C07284=1038.998,375.277,369.594,173.156,44.214,158.680
C07285=1039.007,375.523,369.554,173.163,44.217,158.682
C07286=1039.015,375.770,369.513,173.170,44.221,158.684
C07287=1039.023,376.016,369.472,173.177,44.225,158.685
C07288=1039.032,376.263,369.431,173.184,44.229,158.687
C07289=1039.040,376.510,369.390,173.191,44.233,158.688
C07290=1039.049,376.756,369.350,173.199,44.237,158.690
C07291=1039.062,377.144,369.286,173.210,44.244,158.693
C07292=1039.076,377.532,369.222,173.221,44.250,158.695
C07293=1039.089,377.920,369.157,173.233,44.256,158.698
C07294=1039.103,378.308,369.092,173.244,44.263,158.701
C07295=1039.111,378.555,369.051,173.251,44.266,158.702
C07296=1039.119,378.802,369.011,173.259,44.270,158.704
C07297=1039.128,379.048,368.969,173.266,44.275,158.706
C07298=1039.136,379.295,368.928,173.273,44.279,158.707
C07299=1039.145,379.541,368.886,173.280,44.283,158.709
C07300=1039.153,379.787,368.845,173.288,44.287,158.711
C07301=1039.161,380.034,368.804,173.295,44.291,158.712
C07302=1039.170,380.280,368.762,173.302,44.296,158.714
C07303=1039.178,380.526,368.721,173.309,44.300,158.716
C07304=1039.187,380.773,368.679,173.317,44.304,158.718
C07305=1039.195,381.018,368.638,173.324,44.308,158.719
C07306=1039.204,381.265,368.597,173.331,44.312,158.721
C07307=1039.213,381.512,368.555,173.339,44.317,158.723
C07308=1039.221,381.758,368.514,173.346,44.321,158.725
C07309=1039.230,382.004,368.472,173.354,44.325,158.726
C07310=1039.238,382.251,368.430,173.361,44.329,158.728
C07311=1039.247,382.498,368.389,173.369,44.334,158.730
C07312=1039.255,382.743,368.347,173.376,44.338,158.732
C07313=1039.264,382.990,368.305,173.383,44.343,158.733
C07314=1039.273,383.236,368.264,173.391,44.347,158.735
C07315=1039.281,383.483,368.221,173.399,44.351,158.737
C07316=1039.289,383.728,368.180,173.406,44.355,158.739
C07317=1039.298,383.975,368.138,173.414,44.360,158.741
C07318=1039.307,384.221,368.097,173.421,44.364,158.742
C07319=1039.316,384.467,368.055,173.429,44.369,158.744
C07320=1039.325,384.713,368.012,173.437,44.373,158.746
C07321=1039.334,384.960,367.970,173.445,44.378,158.748
C07322=1039.343,385.206,367.928,173.452,44.382,158.750
C07323=1039.351,385.453,367.887,173.460,44.387,158.752
C07324=1039.360,385.699,367.845,173.468,44.391,158.754
C07325=1039.368,385.944,367.802,173.475,44.395,158.755
C07326=1039.377,386.191,367.761,173.483,44.400,158.757
C07327=1039.386,386.437,367.719,173.491,44.405,158.759
C07328=1039.395,386.683,367.677,173.498,44.409,158.761
C07329=1039.404,386.929,367.634,173.506,44.414,158.763
C07330=1039.413,387.176,367.592,173.515,44.418,158.765
C07331=1039.422,387.422,367.550,173.522,44.423,158.767
C07332=1039.431,387.669,367.508,173.531,44.427,158.769
C07333=1039.440,387.915,367.465,173.538,44.432,158.770
C07334=1039.449,388.161,367.423,173.546,44.437,158.772
C07335=1039.458,388.407,367.381,173.554,44.441,158.774
C07336=1039.466,388.653,367.338,173.562,44.446,158.776
C07337=1039.476,388.899,367.295,173.570,44.450,158.778
C07338=1039.484,389.145,367.253,173.578,44.455,158.780
C07339=1039.493,389.391,367.211,173.585,44.460,158.782
C07340=1039.502,389.638,367.167,173.594,44.464,158.784
C07341=1039.512,389.883,367.125,173.601,44.469,158.786
C07342=1039.520,390.129,367.082,173.610,44.474,158.788
C07343=1039.529,390.376,367.040,173.618,44.479,158.790
C07344=1039.537,390.622,366.997,173.626,44.483,158.792
C07345=1039.547,390.868,366.954,173.634,44.489,158.794
C07346=1039.556,391.114,366.911,173.643,44.493,158.796
C07347=1039.565,391.352,366.870,173.650,44.498,158.798
C07348=1039.573,391.589,366.828,173.658,44.502,158.800
C07349=1039.582,391.827,366.786,173.666,44.507,158.802
C07350=1039.591,392.065,366.745,173.674,44.512,158.804
C07351=1039.599,392.303,366.703,173.682,44.517,158.806
C07352=1039.608,392.541,366.662,173.690,44.521,158.808
C07353=1039.617,392.779,366.620,173.698,44.526,158.809
C07354=1039.626,393.017,366.578,173.707,44.531,158.812
C07355=1039.634,393.263,366.535,173.714,44.536,158.813
C07356=1039.643,393.510,366.492,173.723,44.541,158.816
C07357=1039.653,393.755,366.449,173.732,44.546,158.818
C07358=1039.662,394.001,366.405,173.740,44.551,158.820
C07359=1039.671,394.247,366.362,173.748,44.555,158.822
C07360=1039.681,394.493,366.319,173.756,44.561,158.824
C07361=1039.689,394.739,366.275,173.765,44.566,158.826
C07362=1039.699,394.986,366.232,173.774,44.571,158.828
C07363=1039.708,395.231,366.188,173.783,44.576,158.830
C07364=1039.717,395.477,366.145,173.790,44.581,158.832
C07365=1039.726,395.723,366.101,173.799,44.586,158.834
C07366=1039.735,395.969,366.057,173.808,44.591,158.837
C07367=1039.744,396.214,366.013,173.816,44.596,158.839
C07368=1039.754,396.461,365.971,173.825,44.602,158.841
C07369=1039.763,396.706,365.927,173.834,44.607,158.843
C07370=1039.772,396.952,365.883,173.843,44.612,158.845
C07371=1039.781,397.198,365.839,173.851,44.617,158.847
C07372=1039.790,397.444,365.795,173.860,44.623,158.850
C07373=1039.800,397.690,365.751,173.868,44.628,158.852
C07374=1039.809,397.936,365.707,173.877,44.632,158.854
C07375=1039.819,398.181,365.664,173.886,44.638,158.856
C07376=1039.828,398.427,365.619,173.894,44.643,158.858
C07377=1039.837,398.673,365.576,173.903,44.649,158.861
C07378=1039.846,398.919,365.532,173.912,44.654,158.863
C07379=1039.856,399.165,365.488,173.921,44.659,158.865
C07380=1039.865,399.411,365.443,173.930,44.664,158.867
C07381=1039.875,399.657,365.399,173.939,44.670,158.870
C07382=1039.884,399.903,365.354,173.948,44.675,158.872
C07383=1039.893,400.148,365.311,173.957,44.680,158.874
C07384=1039.903,400.395,365.267,173.966,44.686,158.876
C07385=1039.912,400.640,365.222,173.975,44.691,158.879
C07386=1039.922,400.886,365.178,173.985,44.697,158.881
C07387=1039.931,401.132,365.133,173.994,44.702,158.883
C07388=1039.941,401.378,365.089,174.003,44.708,158.886
C07389=1039.951,401.623,365.044,174.012,44.714,158.888
C07390=1039.960,401.869,365.000,174.021,44.719,158.890
C07391=1039.970,402.115,364.955,174.030,44.725,158.893
C07392=1039.979,402.361,364.910,174.039,44.730,158.895
C07393=1039.989,402.607,364.866,174.049,44.736,158.897
C07394=1039.999,402.852,364.821,174.058,44.741,158.900
C07395=1040.008,403.098,364.776,174.067,44.747,158.902
C07396=1040.017,403.344,364.732,174.076,44.753,158.905
C07397=1040.027,403.590,364.687,174.085,44.758,158.907
C07398=1040.036,403.835,364.642,174.094,44.764,158.909
C07399=1040.045,404.054,364.602,174.103,44.769,158.911
C07400=1040.053,404.274,364.561,174.111,44.774,158.914
C07401=1040.062,404.493,364.521,174.119,44.779,158.916
C07402=1040.071,404.711,364.481,174.128,44.784,158.918
C07403=1040.079,404.930,364.441,174.136,44.789,158.920
C07404=1040.088,405.150,364.400,174.145,44.794,158.922
C07405=1040.096,405.369,364.360,174.153,44.800,158.924
C07406=1040.105,405.588,364.319,174.162,44.805,158.927
C07407=1040.114,405.809,364.279,174.171,44.810,158.929
C07408=1040.122,406.030,364.238,174.179,44.816,158.931
C07409=1040.131,406.251,364.198,174.188,44.820,158.933
C07410=1040.140,406.473,364.157,174.196,44.826,158.936
C07411=1040.149,406.693,364.117,174.205,44.831,158.938
C07412=1040.158,406.914,364.075,174.214,44.837,158.940
C07413=1040.166,407.136,364.034,174.222,44.842,158.942
C07414=1040.175,407.356,363.994,174.231,44.847,158.945
C07415=1040.185,407.602,363.947,174.241,44.853,158.947
C07416=1040.195,407.848,363.902,174.251,44.859,158.950
C07417=1040.205,408.093,363.856,174.261,44.865,158.952
C07418=1040.214,408.339,363.811,174.271,44.871,158.955
C07419=1040.225,408.585,363.765,174.280,44.877,158.957
C07420=1040.235,408.830,363.720,174.290,44.883,158.960
C07421=1040.244,409.076,363.674,174.301,44.889,158.963
C07422=1040.254,409.321,363.628,174.310,44.895,158.965
C07423=1040.265,409.567,363.583,174.321,44.901,158.968
C07424=1040.274,409.812,363.537,174.330,44.907,158.970
C07425=1040.285,410.058,363.491,174.341,44.913,158.973
C07426=1040.295,410.304,363.445,174.350,44.920,158.976
C07427=1040.305,410.549,363.399,174.361,44.925,158.978
C07428=1040.315,410.794,363.353,174.371,44.932,158.981
C07429=1040.325,411.040,363.307,174.381,44.938,158.984
C07430=1040.335,411.285,363.261,174.391,44.944,158.986
C07431=1040.345,411.531,363.215,174.401,44.950,158.989
C07432=1040.356,411.777,363.169,174.412,44.957,158.992
C07433=1040.366,412.023,363.122,174.422,44.963,158.994
C07434=1040.376,412.268,363.076,174.432,44.969,158.997
C07435=1040.386,412.513,363.029,174.442,44.976,159.000
C07436=1040.396,412.759,362.983,174.453,44.982,159.003
C07437=1040.406,413.004,362.937,174.464,44.988,159.005
C07438=1040.416,413.250,362.890,174.473,44.995,159.008
C07439=1040.426,413.496,362.843,174.484,45.001,159.011
C07440=1040.437,413.741,362.796,174.495,45.008,159.014
C07441=1040.447,413.986,362.750,174.506,45.014,159.017
C07442=1040.457,414.232,362.703,174.516,45.020,159.019
C07443=1040.467,414.478,362.656,174.527,45.027,159.022
C07444=1040.478,414.723,362.610,174.537,45.034,159.025
C07445=1040.488,414.968,362.563,174.548,45.040,159.028
C07446=1040.498,415.214,362.516,174.558,45.047,159.031
C07447=1040.508,415.459,362.469,174.569,45.053,159.033
C07448=1040.519,415.704,362.422,174.580,45.060,159.036
C07449=1040.530,415.949,362.375,174.591,45.067,159.039
C07450=1040.540,416.195,362.328,174.602,45.073,159.042
C07451=1040.551,416.440,362.281,174.613,45.080,159.045
C07452=1040.561,416.685,362.234,174.624,45.086,159.048
C07453=1040.571,416.930,362.187,174.635,45.093,159.051
C07454=1040.582,417.176,362.139,174.646,45.099,159.054
C07455=1040.593,417.421,362.093,174.657,45.106,159.057
C07456=1040.603,417.666,362.045,174.668,45.113,159.060
C07457=1040.614,417.912,361.998,174.679,45.120,159.063
C07458=1040.624,418.158,361.951,174.690,45.127,159.066
C07459=1040.634,418.402,361.903,174.701,45.134,159.069
C07460=1040.645,418.648,361.855,174.712,45.141,159.072
C07461=1040.655,418.894,361.808,174.723,45.147,159.075
C07462=1040.666,419.138,361.760,174.735,45.154,159.078
C07463=1040.677,419.384,361.712,174.746,45.161,159.081
C07464=1040.687,419.629,361.664,174.757,45.168,159.084
C07465=1040.698,419.874,361.616,174.769,45.175,159.087
C07466=1040.708,420.120,361.569,174.780,45.182,159.090
C07467=1040.718,420.345,361.525,174.790,45.189,159.093
C07468=1040.728,420.569,361.481,174.801,45.195,159.096
C07469=1040.738,420.795,361.437,174.812,45.201,159.099
C07470=1040.748,421.020,361.393,174.822,45.208,159.102
C07471=1040.758,421.246,361.349,174.833,45.214,159.104
C07472=1040.768,421.470,361.304,174.844,45.221,159.107
C07473=1040.777,421.695,361.261,174.855,45.227,159.110
C07474=1040.788,421.921,361.216,174.865,45.234,159.113
C07475=1040.798,422.165,361.168,174.877,45.241,159.116
C07476=1040.810,422.411,361.119,174.889,45.248,159.119
C07477=1040.821,422.656,361.071,174.900,45.255,159.123
C07478=1040.831,422.901,361.023,174.913,45.262,159.126
C07479=1040.842,423.146,360.975,174.924,45.270,159.129
C07480=1040.853,423.391,360.927,174.937,45.277,159.132
C07481=1040.865,423.636,360.878,174.948,45.284,159.136
C07482=1040.876,423.881,360.829,174.961,45.292,159.139
C07483=1040.887,424.127,360.781,174.972,45.299,159.142
C07484=1040.897,424.371,360.732,174.985,45.307,159.146
C07485=1040.908,424.616,360.683,174.997,45.314,159.149
C07486=1040.920,424.861,360.634,175.009,45.321,159.152
C07487=1040.931,425.107,360.586,175.021,45.329,159.156
C07488=1040.941,425.352,360.537,175.033,45.336,159.159
C07489=1040.953,425.596,360.488,175.046,45.344,159.162
C07490=1040.964,425.841,360.439,175.058,45.351,159.166
C07491=1040.975,426.086,360.390,175.070,45.359,159.169
C07492=1040.986,426.332,360.341,175.083,45.366,159.172
C07493=1040.997,426.576,360.292,175.095,45.374,159.176
C07494=1041.009,426.821,360.243,175.108,45.381,159.179
C07495=1041.020,427.066,360.194,175.120,45.389,159.183
C07496=1041.031,427.311,360.144,175.133,45.397,159.186
C07497=1041.042,427.556,360.095,175.146,45.404,159.190
C07498=1041.054,427.800,360.046,175.158,45.412,159.193
C07499=1041.065,428.046,359.996,175.171,45.420,159.197
C07500=1041.077,428.290,359.946,175.184,45.427,159.200
C07501=1041.088,428.535,359.897,175.197,45.435,159.204
C07502=1041.099,428.780,359.848,175.210,45.443,159.207
C07503=1041.111,429.025,359.798,175.223,45.451,159.211
C07504=1041.122,429.270,359.748,175.236,45.458,159.214
C07505=1041.133,429.514,359.698,175.249,45.466,159.218
C07506=1041.144,429.758,359.648,175.262,45.474,159.222
C07507=1041.156,430.004,359.599,175.275,45.482,159.225
C07508=1041.167,430.248,359.548,175.288,45.490,159.229
C07509=1041.179,430.492,359.498,175.301,45.498,159.232
C07510=1041.191,430.738,359.448,175.314,45.506,159.236
C07511=1041.201,430.983,359.398,175.327,45.515,159.240
C07512=1041.214,431.227,359.348,175.340,45.523,159.243
C07513=1041.225,431.472,359.298,175.354,45.530,159.247
C07514=1041.237,431.717,359.248,175.368,45.539,159.251
C07515=1041.248,431.961,359.197,175.381,45.547,159.255
C07516=1041.260,432.206,359.147,175.394,45.555,159.258
C07517=1041.272,432.450,359.096,175.408,45.563,159.262
C07518=1041.284,432.695,359.046,175.421,45.571,159.266
C07519=1041.295,432.940,358.995,175.435,45.579,159.270
C07520=1041.308,433.185,358.945,175.449,45.588,159.274
C07521=1041.319,433.428,358.894,175.463,45.596,159.277
C07522=1041.331,433.673,358.844,175.477,45.604,159.281
C07523=1041.343,433.918,358.793,175.490,45.613,159.285
C07524=1041.355,434.162,358.743,175.505,45.621,159.289
C07525=1041.367,434.406,358.692,175.518,45.629,159.293
C07526=1041.379,434.651,358.642,175.532,45.637,159.297
C07527=1041.391,434.884,358.593,175.546,45.646,159.301
C07528=1041.402,435.117,358.544,175.559,45.653,159.304
C07529=1041.414,435.351,358.496,175.572,45.662,159.308
C07530=1041.425,435.583,358.447,175.586,45.669,159.312
C07531=1041.437,435.816,358.398,175.600,45.678,159.316
C07532=1041.448,436.049,358.350,175.613,45.686,159.319
C07533=1041.459,436.282,358.300,175.628,45.694,159.323
C07534=1041.471,436.515,358.251,175.641,45.702,159.327
C07535=1041.483,436.759,358.200,175.656,45.711,159.331
C07536=1041.495,437.004,358.149,175.670,45.720,159.335
C07537=1041.508,437.248,358.097,175.684,45.728,159.339
C07538=1041.519,437.492,358.045,175.699,45.737,159.344
C07539=1041.532,437.736,357.994,175.714,45.746,159.348
C07540=1041.544,437.980,357.942,175.728,45.754,159.352
C07541=1041.556,438.225,357.891,175.743,45.763,159.356
C07542=1041.569,438.469,357.838,175.758,45.772,159.360
C07543=1041.581,438.713,357.786,175.773,45.781,159.364
C07544=1041.593,438.958,357.735,175.788,45.789,159.368
C07545=1041.606,439.202,357.682,175.803,45.799,159.373
C07546=1041.619,439.446,357.631,175.818,45.808,159.377
C07547=1041.631,439.690,357.579,175.833,45.817,159.381
C07548=1041.644,439.934,357.526,175.849,45.825,159.386
C07549=1041.656,440.178,357.474,175.864,45.834,159.390
C07550=1041.669,440.423,357.422,175.879,45.844,159.394
C07551=1041.681,440.667,357.370,175.894,45.853,159.399
C07552=1041.694,440.911,357.317,175.910,45.861,159.403
C07553=1041.706,441.155,357.265,175.925,45.871,159.407
C07554=1041.719,441.400,357.212,175.941,45.880,159.412
C07555=1041.731,441.643,357.160,175.957,45.889,159.416
C07556=1041.744,441.888,357.107,175.972,45.898,159.421
C07557=1041.757,442.132,357.054,175.988,45.907,159.425
C07558=1041.769,442.376,357.002,176.004,45.917,159.430
C07559=1041.782,442.620,356.949,176.020,45.926,159.434
C07560=1041.795,442.864,356.896,176.035,45.935,159.439
C07561=1041.808,443.108,356.843,176.052,45.944,159.443
C07562=1041.821,443.352,356.790,176.067,45.954,159.448
C07563=1041.834,443.595,356.737,176.084,45.964,159.452
C07564=1041.846,443.840,356.684,176.100,45.973,159.457
C07565=1041.860,444.084,356.631,176.116,45.982,159.461
C07566=1041.873,444.328,356.578,176.132,45.992,159.466
C07567=1041.886,444.570,356.525,176.149,46.001,159.471
C07568=1041.899,444.814,356.472,176.165,46.011,159.476
C07569=1041.913,445.057,356.419,176.182,46.020,159.480
C07570=1041.927,445.301,356.366,176.199,46.030,159.485
C07571=1041.941,445.544,356.314,176.215,46.039,159.489
C07572=1041.957,445.787,356.263,176.231,46.048,159.494
C07573=1041.972,446.031,356.212,176.248,46.057,159.499
C07574=1041.989,446.275,356.161,176.265,46.066,159.503
C07575=1042.006,446.519,356.111,176.282,46.075,159.508
C07576=1042.023,446.762,356.061,176.299,46.083,159.512
C07577=1042.042,447.006,356.012,176.316,46.092,159.517
C07578=1042.060,447.251,355.963,176.333,46.100,159.521
C07579=1042.080,447.495,355.916,176.351,46.109,159.526
C07580=1042.100,447.740,355.868,176.368,46.117,159.530
C07581=1042.120,447.984,355.820,176.385,46.125,159.535
C07582=1042.141,448.229,355.774,176.402,46.133,159.539
C07583=1042.163,448.473,355.727,176.420,46.141,159.544
C07584=1042.186,448.718,355.681,176.439,46.149,159.548
C07585=1042.209,448.963,355.636,176.455,46.157,159.552
C07586=1042.232,449.208,355.592,176.473,46.165,159.557
C07587=1042.264,449.526,355.534,176.497,46.174,159.562
C07588=1042.296,449.843,355.477,176.520,46.184,159.568
C07589=1042.330,450.161,355.421,176.543,46.193,159.573
C07590=1042.365,450.479,355.367,176.567,46.202,159.579
C07591=1042.392,450.725,355.324,176.586,46.209,159.583
C07592=1042.420,450.970,355.283,176.603,46.216,159.587
C07593=1042.448,451.215,355.242,176.622,46.223,159.592
C07594=1042.477,451.461,355.201,176.641,46.230,159.596
C07595=1042.177,451.505,354.887,176.644,46.308,159.620
C07596=1042.148,451.260,354.927,176.625,46.302,159.616
C07597=1042.119,451.014,354.968,176.606,46.295,159.611
C07598=1042.091,450.768,355.009,176.588,46.289,159.607
C07599=1042.064,450.523,355.051,176.570,46.281,159.603
C07600=1042.031,450.221,355.103,176.546,46.273,159.598
C07601=1041.999,449.918,355.156,176.524,46.264,159.592
C07602=1041.968,449.615,355.210,176.502,46.255,159.587
C07603=1041.937,449.314,355.264,176.480,46.246,159.582
C07604=1041.913,449.069,355.308,176.462,46.238,159.577
C07605=1041.890,448.824,355.354,176.444,46.231,159.573
C07606=1041.867,448.578,355.400,176.427,46.223,159.568
C07607=1041.845,448.334,355.445,176.409,46.215,159.564
C07608=1041.823,448.090,355.492,176.391,46.207,159.560
C07609=1041.803,447.845,355.539,176.373,46.199,159.555
C07610=1041.782,447.601,355.586,176.356,46.191,159.551
C07611=1041.762,447.356,355.634,176.339,46.183,159.546
C07612=1041.743,447.111,355.683,176.321,46.174,159.542
C07613=1041.724,446.868,355.732,176.304,46.166,159.537
C07614=1041.706,446.624,355.781,176.287,46.157,159.533
C07615=1041.689,446.381,355.831,176.270,46.149,159.528
C07616=1041.672,446.136,355.882,176.253,46.140,159.524
C07617=1041.657,445.892,355.932,176.236,46.131,159.519
C07618=1041.641,445.649,355.984,176.219,46.122,159.514
C07619=1041.625,445.406,356.035,176.203,46.113,159.510
C07620=1041.612,445.161,356.087,176.186,46.104,159.505
C07621=1041.597,444.919,356.140,176.170,46.095,159.501
C07622=1041.585,444.675,356.193,176.153,46.085,159.496
C07623=1041.571,444.433,356.245,176.137,46.076,159.491
C07624=1041.558,444.189,356.299,176.120,46.067,159.487
C07625=1041.545,443.945,356.352,176.103,46.057,159.482
C07626=1041.532,443.701,356.405,176.088,46.048,159.477
C07627=1041.519,443.457,356.458,176.072,46.038,159.473
C07628=1041.505,443.213,356.511,176.055,46.029,159.468
C07629=1041.493,442.969,356.564,176.040,46.020,159.464
C07630=1041.480,442.725,356.617,176.023,46.011,159.459
C07631=1041.467,442.481,356.670,176.007,46.001,159.455
C07632=1041.454,442.237,356.723,175.992,45.992,159.450
C07633=1041.441,441.993,356.776,175.975,45.983,159.446
C07634=1041.429,441.749,356.828,175.960,45.974,159.441
C07635=1041.416,441.505,356.881,175.944,45.965,159.437
C07636=1041.403,441.260,356.934,175.928,45.955,159.432
C07637=1041.391,441.017,356.986,175.913,45.946,159.428
C07638=1041.378,440.773,357.039,175.897,45.938,159.424
C07639=1041.366,440.529,357.091,175.882,45.929,159.419
C07640=1041.353,440.284,357.143,175.867,45.920,159.415
C07641=1041.341,440.040,357.196,175.851,45.911,159.411
C07642=1041.328,439.796,357.248,175.836,45.902,159.406
C07643=1041.316,439.552,357.300,175.821,45.893,159.402
C07644=1041.302,439.307,357.352,175.806,45.884,159.398
C07645=1041.290,439.063,357.403,175.791,45.875,159.393
C07646=1041.278,438.819,357.456,175.775,45.866,159.389
C07647=1041.265,438.574,357.508,175.760,45.858,159.385
C07648=1041.253,438.330,357.559,175.745,45.849,159.381
C07649=1041.241,438.086,357.612,175.730,45.840,159.377
C07650=1041.229,437.842,357.663,175.715,45.832,159.373
C07651=1041.216,437.598,357.715,175.700,45.823,159.368
C07652=1041.204,437.353,357.766,175.686,45.814,159.364
C07653=1041.192,437.109,357.818,175.672,45.805,159.360
C07654=1041.180,436.864,357.870,175.657,45.797,159.356
C07655=1041.167,436.620,357.921,175.643,45.789,159.352
C07656=1041.156,436.386,357.970,175.628,45.781,159.348
C07657=1041.144,436.152,358.019,175.615,45.772,159.344
C07658=1041.133,435.919,358.068,175.601,45.764,159.340
C07659=1041.121,435.685,358.117,175.587,45.756,159.336
C07660=1041.110,435.452,358.166,175.574,45.748,159.333
C07661=1041.099,435.218,358.215,175.560,45.740,159.329
C07662=1041.087,434.985,358.264,175.546,45.732,159.325
C07663=1041.075,434.751,358.312,175.533,45.724,159.321
C07664=1041.064,434.506,358.363,175.518,45.716,159.317
C07665=1041.051,434.262,358.414,175.505,45.707,159.314
C07666=1041.039,434.017,358.465,175.491,45.699,159.310
C07667=1041.027,433.773,358.515,175.477,45.691,159.306
C07668=1041.015,433.528,358.566,175.463,45.683,159.302
C07669=1041.003,433.284,358.617,175.449,45.674,159.298
C07670=1040.992,433.039,358.667,175.435,45.666,159.294
C07671=1040.979,432.794,358.717,175.422,45.658,159.290
C07672=1040.968,432.550,358.768,175.407,45.650,159.287
C07673=1040.956,432.305,358.819,175.394,45.642,159.283
C07674=1040.944,432.060,358.869,175.381,45.634,159.279
C07675=1040.932,431.816,358.919,175.367,45.626,159.275
C07676=1040.921,431.571,358.970,175.353,45.618,159.272
C07677=1040.909,431.327,359.019,175.340,45.609,159.268
C07678=1040.898,431.082,359.070,175.327,45.601,159.264
C07679=1040.886,430.838,359.120,175.313,45.594,159.260
C07680=1040.874,430.593,359.170,175.300,45.586,159.257
C07681=1040.863,430.348,359.220,175.287,45.578,159.253
C07682=1040.851,430.103,359.270,175.274,45.570,159.250
C07683=1040.840,429.859,359.320,175.261,45.562,159.246
C07684=1040.829,429.614,359.370,175.248,45.554,159.242
C07685=1040.817,429.369,359.420,175.235,45.546,159.239
C07686=1040.806,429.124,359.470,175.221,45.538,159.235
C07687=1040.794,428.880,359.520,175.209,45.531,159.232
C07688=1040.783,428.634,359.570,175.196,45.523,159.228
C07689=1040.771,428.390,359.619,175.183,45.516,159.224
C07690=1040.760,428.145,359.669,175.170,45.508,159.221
C07691=1040.749,427.900,359.718,175.157,45.500,159.217
C07692=1040.737,427.656,359.767,175.144,45.492,159.214
C07693=1040.726,427.410,359.817,175.131,45.485,159.210
C07694=1040.715,427.165,359.866,175.119,45.477,159.207
C07695=1040.703,426.920,359.915,175.106,45.470,159.203
C07696=1040.692,426.676,359.964,175.093,45.462,159.200
C07697=1040.681,426.431,360.014,175.081,45.455,159.197
C07698=1040.670,426.186,360.063,175.069,45.447,159.193
C07699=1040.658,425.941,360.112,175.056,45.440,159.190
C07700=1040.647,425.696,360.161,175.043,45.432,159.186
C07701=1040.636,425.451,360.210,175.031,45.425,159.183
C07702=1040.625,425.206,360.259,175.019,45.417,159.180
C07703=1040.614,424.961,360.308,175.006,45.410,159.176
C07704=1040.602,424.717,360.357,174.995,45.402,159.173
C07705=1040.592,424.471,360.405,174.982,45.396,159.170
C07706=1040.581,424.227,360.454,174.969,45.388,159.166
C07707=1040.570,423.982,360.502,174.958,45.381,159.163
C07708=1040.559,423.737,360.551,174.945,45.373,159.160
C07709=1040.548,423.491,360.600,174.934,45.366,159.156
C07710=1040.537,423.246,360.648,174.921,45.359,159.153
C07711=1040.526,423.001,360.696,174.910,45.352,159.150
C07712=1040.515,422.757,360.745,174.898,45.345,159.147
C07713=1040.504,422.511,360.793,174.886,45.338,159.144
C07714=1040.493,422.266,360.842,174.874,45.331,159.140
C07715=1040.482,422.021,360.890,174.862,45.324,159.137
C07716=1040.472,421.794,360.935,174.851,45.317,159.134
C07717=1040.462,421.569,360.979,174.840,45.310,159.131
C07718=1040.452,421.343,361.023,174.830,45.304,159.128
C07719=1040.442,421.115,361.067,174.819,45.297,159.125
C07720=1040.432,420.890,361.111,174.808,45.291,159.123
C07721=1040.422,420.663,361.156,174.797,45.284,159.120
C07722=1040.411,420.437,361.200,174.787,45.278,159.117
C07723=1040.402,420.210,361.244,174.776,45.272,159.114
C07724=1040.392,419.965,361.292,174.765,45.264,159.111
C07725=1040.381,419.720,361.341,174.753,45.258,159.108
C07726=1040.370,419.475,361.388,174.742,45.251,159.105
C07727=1040.359,419.229,361.436,174.730,45.244,159.102
C07728=1040.349,418.984,361.483,174.719,45.237,159.099
C07729=1040.339,418.740,361.531,174.708,45.231,159.096
C07730=1040.328,418.494,361.579,174.697,45.223,159.093
C07731=1040.318,418.248,361.626,174.686,45.217,159.090
C07732=1040.307,418.004,361.674,174.674,45.210,159.087
C07733=1040.296,417.758,361.722,174.663,45.203,159.084
C07734=1040.285,417.513,361.768,174.652,45.197,159.081
C07735=1040.275,417.267,361.815,174.640,45.190,159.078
C07736=1040.264,417.021,361.863,174.630,45.184,159.075
C07737=1040.254,416.776,361.910,174.619,45.177,159.072
C07738=1040.243,416.531,361.957,174.607,45.170,159.069
C07739=1040.233,416.286,362.004,174.597,45.164,159.066
C07740=1040.223,416.041,362.051,174.586,45.157,159.063
C07741=1040.212,415.796,362.098,174.575,45.150,159.060
C07742=1040.201,415.550,362.146,174.565,45.144,159.057
C07743=1040.191,415.304,362.193,174.554,45.137,159.054
C07744=1040.181,415.059,362.240,174.543,45.131,159.052
C07745=1040.170,414.813,362.286,174.532,45.125,159.049
C07746=1040.160,414.568,362.333,174.521,45.118,159.046
C07747=1040.150,414.323,362.380,174.510,45.112,159.043
C07748=1040.139,414.077,362.426,174.499,45.105,159.040
C07749=1040.129,413.832,362.473,174.490,45.099,159.038
C07750=1040.120,413.587,362.520,174.479,45.093,159.035
C07751=1040.109,413.342,362.566,174.468,45.086,159.032
C07752=1040.099,413.096,362.613,174.457,45.079,159.029
C07753=1040.089,412.851,362.660,174.447,45.073,159.026
C07754=1040.079,412.605,362.706,174.437,45.067,159.024
C07755=1040.068,412.360,362.753,174.426,45.061,159.021
C07756=1040.059,412.115,362.799,174.416,45.054,159.018
C07757=1040.049,411.869,362.846,174.406,45.048,159.015
C07758=1040.038,411.623,362.892,174.395,45.042,159.013
C07759=1040.028,411.377,362.938,174.385,45.036,159.010
C07760=1040.018,411.132,362.984,174.374,45.030,159.007
C07761=1040.008,410.887,363.030,174.365,45.023,159.005
C07762=1039.998,410.641,363.076,174.354,45.017,159.002
C07763=1039.987,410.395,363.122,174.344,45.011,158.999
C07764=1039.977,410.150,363.168,174.334,45.005,158.997
C07765=1039.967,409.904,363.214,174.324,44.999,158.994
C07766=1039.957,409.659,363.260,174.314,44.993,158.991
C07767=1039.947,409.414,363.305,174.303,44.987,158.989
C07768=1039.937,409.167,363.351,174.294,44.981,158.986
C07769=1039.926,408.922,363.397,174.283,44.975,158.984
C07770=1039.917,408.677,363.443,174.274,44.969,158.981
C07771=1039.907,408.430,363.488,174.263,44.963,158.978
C07772=1039.897,408.185,363.534,174.254,44.957,158.976
C07773=1039.887,407.939,363.580,174.244,44.951,158.973
C07774=1039.877,407.694,363.625,174.234,44.945,158.971
C07775=1039.867,407.448,363.670,174.224,44.939,158.968
C07776=1039.858,407.226,363.712,174.215,44.934,158.966
C07777=1039.849,407.004,363.753,174.206,44.929,158.964
C07778=1039.840,406.782,363.794,174.198,44.924,158.962
C07779=1039.831,406.559,363.835,174.189,44.918,158.959
C07780=1039.823,406.338,363.876,174.180,44.913,158.957
C07781=1039.814,406.116,363.917,174.172,44.908,158.955
C07782=1039.805,405.893,363.958,174.163,44.902,158.952
C07783=1039.796,405.671,363.999,174.154,44.897,158.950
C07784=1039.787,405.425,364.045,174.144,44.891,158.948
C07785=1039.777,405.179,364.089,174.135,44.886,158.945
C07786=1039.767,404.934,364.134,174.126,44.880,158.943
C07787=1039.758,404.688,364.180,174.116,44.875,158.940
C07788=1039.749,404.443,364.225,174.106,44.869,158.938
C07789=1039.738,404.197,364.270,174.097,44.863,158.936
C07790=1039.729,403.951,364.315,174.088,44.858,158.933
C07791=1039.720,403.705,364.360,174.078,44.852,158.931
C07792=1039.710,403.459,364.405,174.069,44.846,158.928
C07793=1039.700,403.214,364.450,174.060,44.841,158.926
C07794=1039.691,402.968,364.495,174.050,44.835,158.924
C07795=1039.681,402.723,364.540,174.041,44.829,158.921
C07796=1039.672,402.477,364.584,174.031,44.824,158.919
C07797=1039.662,402.231,364.629,174.022,44.818,158.916
C07798=1039.653,401.985,364.674,174.013,44.813,158.914
C07799=1039.643,401.739,364.718,174.004,44.807,158.912
C07800=1039.633,401.494,364.763,173.995,44.802,158.909
C07801=1039.624,401.248,364.807,173.986,44.797,158.907
C07802=1039.614,401.002,364.851,173.977,44.791,158.905
C07803=1039.605,400.756,364.896,173.968,44.786,158.903
C07804=1039.595,400.511,364.940,173.958,44.780,158.900
C07805=1039.586,400.264,364.984,173.949,44.775,158.898
C07806=1039.576,400.018,365.029,173.940,44.770,158.896
C07807=1039.567,399.773,365.073,173.931,44.764,158.893
C07808=1039.558,399.527,365.117,173.922,44.759,158.891
C07809=1039.548,399.281,365.161,173.913,44.754,158.889
C07810=1039.539,399.035,365.205,173.904,44.748,158.887
C07811=1039.529,398.790,365.250,173.895,44.743,158.884
C07812=1039.520,398.544,365.294,173.886,44.738,158.882
C07813=1039.511,398.298,365.338,173.878,44.733,158.880
C07814=1039.501,398.052,365.382,173.869,44.728,158.878
C07815=1039.492,397.806,365.426,173.861,44.723,158.876
C07816=1039.483,397.561,365.469,173.851,44.717,158.873
C07817=1039.473,397.314,365.514,173.843,44.712,158.871
C07818=1039.464,397.068,365.558,173.834,44.707,158.869
C07819=1039.455,396.823,365.601,173.826,44.702,158.867
C07820=1039.446,396.576,365.645,173.817,44.696,158.865
C07821=1039.436,396.331,365.688,173.808,44.691,158.862
C07822=1039.427,396.085,365.732,173.799,44.686,158.860
C07823=1039.418,395.839,365.776,173.790,44.681,158.858
C07824=1039.409,395.593,365.819,173.782,44.676,158.856
C07825=1039.400,395.347,365.863,173.773,44.671,158.854
C07826=1039.390,395.101,365.906,173.765,44.666,158.852
C07827=1039.381,394.855,365.950,173.757,44.661,158.850
C07828=1039.372,394.609,365.994,173.748,44.656,158.848
C07829=1039.362,394.363,366.036,173.739,44.651,158.846
C07830=1039.354,394.117,366.080,173.730,44.646,158.843
C07831=1039.345,393.871,366.123,173.723,44.641,158.841
C07832=1039.334,393.573,366.176,173.712,44.635,158.839
C07833=1039.323,393.275,366.228,173.702,44.629,158.836
C07834=1039.312,392.977,366.280,173.691,44.623,158.834
C07835=1039.300,392.680,366.333,173.681,44.618,158.831
C07836=1039.287,392.307,366.398,173.669,44.611,158.828
C07837=1039.273,391.934,366.464,173.657,44.603,158.825
C07838=1039.259,391.562,366.528,173.644,44.596,158.822
C07839=1039.246,391.189,366.593,173.632,44.588,158.819
C07840=1039.237,390.943,366.636,173.623,44.584,158.817
C07841=1039.228,390.696,366.680,173.616,44.579,158.815
C07842=1039.219,390.451,366.722,173.607,44.574,158.813
C07843=1039.210,390.205,366.765,173.599,44.569,158.811
C07844=1039.201,389.959,366.808,173.591,44.565,158.809
C07845=1039.192,389.713,366.849,173.583,44.560,158.807
C07846=1039.183,389.466,366.893,173.575,44.556,158.805
C07847=1039.174,389.220,366.935,173.567,44.551,158.803
C07848=1039.165,388.974,366.978,173.559,44.547,158.801
C07849=1039.156,388.728,367.021,173.551,44.541,158.799
C07850=1039.148,388.482,367.063,173.542,44.537,158.797
C07851=1039.139,388.236,367.105,173.535,44.533,158.796
C07852=1039.130,387.990,367.148,173.526,44.528,158.794
C07853=1039.121,387.743,367.190,173.519,44.523,158.792
C07854=1039.112,387.498,367.233,173.511,44.519,158.790
C07855=1039.103,387.250,367.275,173.503,44.514,158.788
C07856=1039.094,387.005,367.318,173.495,44.510,158.786
C07857=1039.085,386.758,367.359,173.487,44.506,158.784
C07858=1039.076,386.512,367.401,173.479,44.501,158.782
C07859=1039.067,386.266,367.444,173.472,44.496,158.780
C07860=1039.059,386.019,367.486,173.463,44.492,158.779
C07861=1039.050,385.773,367.528,173.456,44.488,158.777
C07862=1039.040,385.527,367.570,173.448,44.483,158.775
C07863=1039.031,385.281,367.612,173.440,44.479,158.773
C07864=1039.023,385.035,367.653,173.432,44.474,158.771
C07865=1039.015,384.789,367.695,173.425,44.470,158.769
C07866=1039.006,384.542,367.737,173.418,44.466,158.768
C07867=1038.997,384.296,367.779,173.409,44.461,158.766
C07868=1038.988,384.050,367.821,173.402,44.457,158.764
C07869=1038.979,383.804,367.863,173.394,44.452,158.762
C07870=1038.971,383.557,367.905,173.386,44.449,158.760
C07871=1038.962,383.311,367.947,173.379,44.444,158.759
C07872=1038.953,383.065,367.988,173.371,44.440,158.757
C07873=1038.944,382.819,368.030,173.364,44.435,158.755
C07874=1038.936,382.572,368.072,173.357,44.431,158.753
C07875=1038.927,382.326,368.114,173.348,44.427,158.751
C07876=1038.919,382.079,368.155,173.341,44.423,158.750
C07877=1038.910,381.833,368.196,173.334,44.418,158.748
C07878=1038.901,381.587,368.238,173.326,44.414,158.746
C07879=1038.893,381.341,368.279,173.319,44.410,158.744
C07880=1038.884,381.095,368.321,173.312,44.406,158.743
C07881=1038.876,380.847,368.363,173.305,44.402,158.741
C07882=1038.868,380.602,368.404,173.296,44.398,158.739
C07883=1038.859,380.355,368.446,173.289,44.394,158.737
C07884=1038.850,380.108,368.487,173.282,44.389,158.736
C07885=1038.842,379.863,368.528,173.274,44.385,158.734
C07886=1038.833,379.616,368.569,173.267,44.381,158.732
C07887=1038.826,379.370,368.611,173.260,44.377,158.731
C07888=1038.817,379.123,368.653,173.253,44.373,158.729
C07889=1038.809,378.877,368.693,173.245,44.368,158.727
C07890=1038.800,378.631,368.735,173.238,44.365,158.726
C07891=1038.792,378.384,368.776,173.231,44.361,158.724
C07892=1038.778,377.994,368.841,173.220,44.354,158.721
C07893=1038.765,377.603,368.906,173.208,44.348,158.718
C07894=1038.751,377.214,368.970,173.197,44.342,158.716
C07895=1038.738,376.823,369.035,173.185,44.335,158.713
C07896=1038.730,376.576,369.075,173.178,44.332,158.712
C07897=1038.721,376.330,369.117,173.171,44.327,158.710
C07898=1038.712,376.084,369.157,173.164,44.324,158.708
C07899=1038.703,375.837,369.198,173.157,44.320,158.707
C07900=1038.695,375.591,369.239,173.150,44.316,158.705
C07901=1038.687,375.344,369.280,173.143,44.312,158.704
C07902=1038.679,375.098,369.320,173.135,44.308,158.702
C07903=1038.671,374.851,369.361,173.128,44.304,158.700
C07904=1038.661,374.605,369.401,173.121,44.301,158.699
C07905=1038.653,374.358,369.442,173.114,44.297,158.697
C07906=1038.646,374.111,369.482,173.107,44.293,158.696
C07907=1038.637,373.864,369.523,173.101,44.289,158.694
C07908=1038.629,373.618,369.564,173.094,44.285,158.693
C07909=1038.620,373.372,369.604,173.087,44.282,158.691
C07910=1038.612,373.126,369.644,173.080,44.278,158.689
C07911=1038.604,372.878,369.685,173.073,44.274,158.688
C07912=1038.596,372.632,369.725,173.066,44.270,158.686
C07913=1038.588,372.386,369.766,173.059,44.267,158.685
C07914=1038.579,372.139,369.805,173.053,44.263,158.683
C07915=1038.571,371.893,369.846,173.046,44.259,158.682
C07916=1038.563,371.646,369.887,173.039,44.255,158.680
C07917=1038.555,371.399,369.927,173.032,44.252,158.679
C07918=1038.546,371.153,369.967,173.025,44.248,158.677
C07919=1038.538,370.906,370.007,173.019,44.244,158.675
C07920=1038.530,370.660,370.047,173.012,44.241,158.674
C07921=1038.523,370.413,370.087,173.005,44.237,158.672
C07922=1038.515,370.167,370.128,172.998,44.233,158.671
C07923=1038.506,369.920,370.167,172.992,44.229,158.669
C07924=1038.497,369.673,370.207,172.985,44.226,158.668
C07925=1038.489,369.426,370.248,172.978,44.223,158.666
C07926=1038.481,369.180,370.287,172.971,44.219,158.665
C07927=1038.473,368.933,370.327,172.964,44.215,158.663
C07928=1038.464,368.686,370.366,172.959,44.212,158.662
C07929=1038.456,368.440,370.407,172.952,44.208,158.661
C07930=1038.448,368.193,370.446,172.945,44.205,158.659
C07931=1038.440,367.946,370.486,172.939,44.201,158.658
C07932=1038.432,367.700,370.525,172.932,44.198,158.656
C07933=1038.424,367.453,370.565,172.925,44.195,158.655
C07934=1038.416,367.206,370.605,172.918,44.191,158.653
C07935=1038.408,366.959,370.645,172.912,44.188,158.652
C07936=1038.399,366.713,370.684,172.905,44.184,158.650
C07937=1038.391,366.466,370.723,172.899,44.181,158.649
C07938=1038.383,366.219,370.763,172.893,44.177,158.647
C07939=1038.375,365.973,370.802,172.886,44.174,158.646
C07940=1038.367,365.726,370.842,172.880,44.171,158.645
C07941=1038.359,365.479,370.882,172.873,44.167,158.643
C07942=1038.351,365.232,370.922,172.867,44.164,158.642
C07943=1038.343,364.987,370.961,172.861,44.160,158.640
C07944=1038.336,364.739,371.000,172.854,44.157,158.639
C07945=1038.327,364.492,371.039,172.847,44.154,158.638
C07946=1038.319,364.246,371.078,172.841,44.150,158.636
C07947=1038.311,363.999,371.118,172.834,44.147,158.635
C07948=1038.299,363.629,371.177,172.825,44.142,158.633
C07949=1038.287,363.259,371.236,172.816,44.137,158.631
C07950=1038.276,362.889,371.294,172.807,44.132,158.629
C07951=1038.264,362.519,371.353,172.797,44.127,158.627
C07952=1038.256,362.271,371.392,172.790,44.124,158.625
C07953=1038.248,362.025,371.432,172.784,44.120,158.624
C07954=1038.240,361.778,371.470,172.778,44.117,158.623
C07955=1038.232,361.531,371.510,172.772,44.114,158.621
C07956=1038.224,361.284,371.549,172.765,44.111,158.620
C07957=1038.216,361.037,371.587,172.760,44.108,158.619
C07958=1038.208,360.791,371.626,172.753,44.104,158.617
C07959=1038.200,360.544,371.665,172.747,44.101,158.616
C07960=1038.192,360.297,371.703,172.740,44.098,158.615
C07961=1038.185,360.050,371.743,172.735,44.095,158.613
C07962=1038.177,359.803,371.782,172.728,44.091,158.612
C07963=1038.169,359.556,371.820,172.722,44.089,158.611
C07964=1038.161,359.309,371.858,172.716,44.086,158.609
C07965=1038.152,359.063,371.898,172.710,44.082,158.608
C07966=1038.145,358.816,371.936,172.704,44.079,158.607
C07967=1038.137,358.569,371.975,172.698,44.076,158.606
C07968=1038.129,358.322,372.013,172.692,44.073,158.604
C07969=1038.121,358.075,372.051,172.685,44.070,158.603
C07970=1038.114,357.828,372.091,172.680,44.067,158.602
C07971=1038.106,357.581,372.129,172.673,44.064,158.600
C07972=1038.098,357.334,372.167,172.667,44.061,158.599
C07973=1038.090,357.088,372.206,172.662,44.058,158.598
C07974=1038.082,356.840,372.244,172.655,44.055,158.597
C07975=1038.075,356.594,372.283,172.650,44.051,158.595
C07976=1038.067,356.347,372.321,172.644,44.049,158.594
C07977=1038.059,356.100,372.359,172.637,44.046,158.593
C07978=1038.051,355.853,372.398,172.632,44.043,158.592
C07979=1038.044,355.606,372.436,172.625,44.040,158.590
C07980=1038.035,355.359,372.474,172.620,44.037,158.589
C07981=1038.028,355.112,372.512,172.614,44.034,158.588
C07982=1038.020,354.865,372.551,172.608,44.031,158.587
C07983=1038.012,354.618,372.588,172.602,44.028,158.585
C07984=1038.004,354.371,372.626,172.596,44.025,158.584
C07985=1037.996,354.124,372.665,172.590,44.022,158.583
C07986=1037.989,353.877,372.702,172.584,44.020,158.582
C07987=1037.981,353.630,372.741,172.579,44.016,158.581
C07988=1037.973,353.383,372.779,172.572,44.014,158.579
C07989=1037.966,353.136,372.817,172.567,44.011,158.578
C07990=1037.958,352.889,372.855,172.561,44.008,158.577
C07991=1037.950,352.642,372.892,172.555,44.005,158.576
C07992=1037.942,352.396,372.930,172.549,44.002,158.575
C07993=1037.934,352.148,372.968,172.544,43.999,158.573
C07994=1037.927,351.901,373.007,172.538,43.996,158.572
C07995=1037.920,351.654,373.044,172.532,43.994,158.571
C07996=1037.912,351.408,373.082,172.526,43.991,158.570
C07997=1037.904,351.160,373.120,172.521,43.988,158.569
C07998=1037.897,350.913,373.158,172.515,43.985,158.567
C07999=1037.889,350.667,373.195,172.509,43.983,158.566
C08000=1037.881,350.419,373.233,172.503,43.980,158.565
C08001=1037.874,350.172,373.271,172.498,43.977,158.564
C08002=1037.866,349.925,373.309,172.492,43.974,158.563
C08003=1037.859,349.678,373.347,172.487,43.971,158.562
C08004=1037.847,349.314,373.402,172.478,43.968,158.560
C08005=1037.836,348.950,373.457,172.470,43.963,158.558
C08006=1037.825,348.586,373.512,172.461,43.959,158.557
C08007=1037.814,348.221,373.568,172.453,43.955,158.555
C08008=1037.806,347.974,373.605,172.448,43.953,158.554
C08009=1037.798,347.727,373.642,172.442,43.950,158.553
C08010=1037.790,347.480,373.679,172.436,43.948,158.552
C08011=1037.783,347.233,373.717,172.431,43.945,158.550
C08012=1037.776,346.986,373.754,172.425,43.942,158.549
C08013=1037.768,346.739,373.791,172.420,43.939,158.548
C08014=1037.761,346.492,373.829,172.415,43.937,158.547
C08015=1037.753,346.245,373.866,172.409,43.934,158.546
C08016=1037.745,345.998,373.903,172.403,43.932,158.545
C08017=1037.738,345.751,373.941,172.397,43.929,158.544
C08018=1037.730,345.504,373.978,172.392,43.927,158.543
C08019=1037.723,345.256,374.015,172.387,43.924,158.542
C08020=1037.715,345.009,374.052,172.381,43.921,158.540
C08021=1037.707,344.762,374.089,172.376,43.919,158.539
C08022=1037.699,344.515,374.126,172.370,43.916,158.538
C08023=1037.692,344.267,374.163,172.365,43.914,158.537
C08024=1037.684,344.020,374.200,172.360,43.911,158.536
C08025=1037.677,343.773,374.237,172.354,43.908,158.535
C08026=1037.670,343.527,374.274,172.348,43.906,158.534
C08027=1037.663,343.279,374.311,172.343,43.903,158.533
C08028=1037.655,343.033,374.348,172.337,43.901,158.532
C08029=1037.648,342.785,374.384,172.332,43.898,158.531
C08030=1037.640,342.538,374.421,172.327,43.896,158.530
C08031=1037.633,342.291,374.459,172.321,43.893,158.529
C08032=1037.625,342.043,374.495,172.316,43.891,158.528
C08033=1037.618,341.796,374.533,172.311,43.888,158.527
C08034=1037.610,341.549,374.569,172.305,43.886,158.526
C08035=1037.603,341.302,374.606,172.300,43.883,158.525
C08036=1037.596,341.055,374.642,172.295,43.881,158.524
C08037=1037.588,340.808,374.678,172.290,43.879,158.523
C08038=1037.580,340.561,374.715,172.284,43.876,158.521
C08039=1037.573,340.313,374.752,172.279,43.874,158.520
C08040=1037.566,340.065,374.788,172.274,43.872,158.519
C08041=1037.558,339.819,374.825,172.269,43.870,158.519
C08042=1037.550,339.571,374.862,172.263,43.867,158.517
C08043=1037.544,339.324,374.898,172.258,43.865,158.516
C08044=1037.536,339.077,374.934,172.253,43.862,158.515
C08045=1037.528,338.830,374.971,172.248,43.860,158.514
C08046=1037.520,338.582,375.007,172.242,43.857,158.513
C08047=1037.513,338.335,375.044,172.237,43.855,158.512
C08048=1037.506,338.088,375.080,172.232,43.853,158.511
C08049=1037.499,337.841,375.116,172.226,43.851,158.510
C08050=1037.491,337.593,375.153,172.221,43.848,158.509
C08051=1037.485,337.346,375.189,172.216,43.846,158.508
C08052=1037.477,337.099,375.226,172.211,43.843,158.507
C08053=1037.469,336.852,375.262,172.205,43.841,158.506
C08054=1037.461,336.604,375.298,172.200,43.839,158.505
C08055=1037.455,336.357,375.335,172.196,43.837,158.504
C08056=1037.447,336.110,375.371,172.191,43.834,158.504
C08057=1037.440,335.862,375.407,172.186,43.832,158.503
C08058=1037.432,335.616,375.443,172.180,43.830,158.502
C08059=1037.425,335.368,375.479,172.175,43.828,158.501
C08060=1037.414,335.000,375.533,172.168,43.825,158.499
C08061=1037.404,334.633,375.586,172.160,43.821,158.498
C08062=1037.393,334.266,375.640,172.153,43.818,158.496
C08063=1037.382,333.898,375.694,172.145,43.815,158.495
C08064=1037.374,333.650,375.729,172.140,43.813,158.494
C08065=1037.367,333.403,375.764,172.135,43.810,158.493
C08066=1037.359,333.156,375.801,172.130,43.808,158.492
C08067=1037.352,332.908,375.836,172.124,43.806,158.491
C08068=1037.344,332.661,375.872,172.120,43.803,158.490
C08069=1037.337,332.414,375.908,172.115,43.802,158.489
C08070=1037.330,332.166,375.943,172.110,43.800,158.488
C08071=1037.323,331.919,375.979,172.105,43.797,158.488
C08072=1037.315,331.672,376.015,172.100,43.795,158.487
C08073=1037.308,331.425,376.051,172.095,43.793,158.486
C08074=1037.301,331.177,376.087,172.090,43.791,158.485
C08075=1037.294,330.930,376.122,172.085,43.789,158.484
C08076=1037.286,330.682,376.158,172.080,43.787,158.483
C08077=1037.280,330.435,376.193,172.075,43.785,158.482
C08078=1037.272,330.188,376.230,172.070,43.783,158.481
C08079=1037.265,329.940,376.265,172.065,43.780,158.480
C08080=1037.257,329.693,376.301,172.061,43.779,158.479
C08081=1037.251,329.445,376.336,172.056,43.776,158.478
C08082=1037.243,329.198,376.372,172.051,43.774,158.477
C08083=1037.236,328.951,376.407,172.046,43.773,158.477
C08084=1037.229,328.703,376.442,172.041,43.770,158.476
C08085=1037.221,328.456,376.478,172.036,43.768,158.475
C08086=1037.214,328.209,376.513,172.031,43.766,158.474
C08087=1037.207,327.961,376.549,172.026,43.765,158.473
C08088=1037.199,327.714,376.583,172.021,43.762,158.472
C08089=1037.192,327.466,376.619,172.017,43.761,158.471
C08090=1037.184,327.219,376.654,172.012,43.758,158.470
C08091=1037.177,326.972,376.689,172.007,43.757,158.470
C08092=1037.169,326.724,376.724,172.002,43.755,158.469
C08093=1037.163,326.477,376.759,171.998,43.753,158.468
C08094=1037.155,326.230,376.794,171.993,43.751,158.467
C08095=1037.148,325.981,376.829,171.988,43.749,158.466
C08096=1037.140,325.734,376.864,171.983,43.747,158.465
C08097=1037.133,325.486,376.899,171.979,43.745,158.465
C08098=1037.125,325.239,376.934,171.974,43.744,158.464
C08099=1037.119,324.992,376.969,171.969,43.741,158.463
C08100=1037.111,324.745,377.004,171.964,43.740,158.462
C08101=1037.104,324.497,377.039,171.960,43.738,158.461
C08102=1037.096,324.250,377.074,171.955,43.736,158.461
C08103=1037.089,324.002,377.109,171.950,43.734,158.460
C08104=1037.081,323.755,377.144,171.946,43.732,158.459
C08105=1037.075,323.507,377.179,171.941,43.730,158.458
C08106=1037.068,323.260,377.214,171.936,43.729,158.457
C08107=1037.061,323.012,377.248,171.931,43.727,158.456
C08108=1037.053,322.764,377.283,171.927,43.725,158.455
C08109=1037.046,322.517,377.318,171.922,43.723,158.455
C08110=1037.039,322.270,377.353,171.917,43.721,158.454
C08111=1037.031,322.023,377.387,171.913,43.720,158.453
C08112=1037.024,321.776,377.422,171.908,43.717,158.452
C08113=1037.017,321.527,377.457,171.903,43.716,158.451
C08114=1037.009,321.280,377.491,171.899,43.714,158.451
C08115=1037.003,321.033,377.526,171.894,43.712,158.450
C08116=1036.992,320.661,377.579,171.887,43.709,158.449
C08117=1036.981,320.288,377.631,171.880,43.707,158.447
C08118=1036.971,319.916,377.683,171.873,43.704,158.446
C08119=1036.959,319.544,377.735,171.866,43.701,158.445
C08120=1036.953,319.296,377.769,171.862,43.699,158.444
C08121=1036.945,319.049,377.804,171.857,43.698,158.443
C08122=1036.939,318.801,377.839,171.853,43.696,158.443
C08123=1036.931,318.554,377.873,171.848,43.694,158.442
C08124=1036.925,318.306,377.908,171.843,43.693,158.441
C08125=1036.917,318.059,377.942,171.839,43.691,158.440
C08126=1036.911,317.811,377.977,171.834,43.689,158.439
C08127=1036.903,317.564,378.010,171.830,43.687,158.439
C08128=1036.896,317.316,378.045,171.825,43.686,158.438
C08129=1036.889,317.068,378.079,171.820,43.684,158.437
C08130=1036.882,316.821,378.114,171.816,43.682,158.436
C08131=1036.876,316.573,378.148,171.811,43.680,158.436
C08132=1036.868,316.326,378.182,171.807,43.678,158.435
C08133=1036.862,316.078,378.217,171.802,43.677,158.434
C08134=1036.855,315.831,378.251,171.799,43.675,158.433
C08135=1036.848,315.584,378.286,171.794,43.673,158.432
C08136=1036.841,315.336,378.320,171.790,43.672,158.432
C08137=1036.834,315.089,378.354,171.785,43.670,158.431
C08138=1036.827,314.841,378.389,171.781,43.669,158.430
C08139=1036.820,314.594,378.423,171.776,43.667,158.429
C08140=1036.813,314.346,378.457,171.772,43.665,158.429
C08141=1036.806,314.098,378.491,171.767,43.663,158.428
C08142=1036.800,313.851,378.526,171.763,43.661,158.427
C08143=1036.793,313.604,378.559,171.758,43.660,158.426
C08144=1036.786,313.356,378.593,171.755,43.659,158.426
C08145=1036.779,313.108,378.628,171.750,43.657,158.425
C08146=1036.772,312.861,378.662,171.746,43.655,158.424
C08147=1036.766,312.614,378.696,171.741,43.653,158.423
C08148=1036.759,312.366,378.730,171.737,43.651,158.423
C08149=1036.751,312.118,378.764,171.732,43.650,158.422
C08150=1036.745,311.870,378.798,171.728,43.649,158.421
C08151=1036.738,311.623,378.832,171.723,43.647,158.420
C08152=1036.730,311.375,378.866,171.719,43.646,158.420
C08153=1036.724,311.128,378.899,171.714,43.644,158.419
C08154=1036.716,310.881,378.933,171.711,43.642,158.418
C08155=1036.709,310.633,378.966,171.706,43.641,158.418
C08156=1036.702,310.385,379.000,171.702,43.639,158.417
C08157=1036.694,310.138,379.034,171.697,43.638,158.416
C08158=1036.687,309.889,379.067,171.693,43.636,158.416
C08159=1036.681,309.642,379.101,171.689,43.635,158.415
C08160=1036.673,309.395,379.134,171.685,43.633,158.414
C08161=1036.666,309.147,379.168,171.680,43.632,158.414
C08162=1036.659,308.900,379.202,171.676,43.631,158.413
C08163=1036.652,308.652,379.234,171.672,43.629,158.412
C08164=1036.645,308.404,379.268,171.667,43.628,158.412
C08165=1036.637,308.157,379.301,171.664,43.626,158.411
C08166=1036.630,307.909,379.334,171.659,43.625,158.410
C08167=1036.624,307.662,379.368,171.655,43.623,158.409
C08168=1036.616,307.414,379.402,171.650,43.622,158.409
C08169=1036.609,307.166,379.436,171.646,43.621,158.408
C08170=1036.602,306.918,379.469,171.642,43.619,158.407
C08171=1036.595,306.671,379.502,171.638,43.618,158.407
C08172=1036.585,306.304,379.551,171.632,43.616,158.406
C08173=1036.574,305.936,379.601,171.625,43.614,158.405
C08174=1036.563,305.569,379.650,171.619,43.612,158.404
C08175=1036.553,305.201,379.699,171.613,43.610,158.403
C08176=1036.547,304.954,379.732,171.608,43.608,158.402
C08177=1036.540,304.706,379.766,171.604,43.607,158.401
C08178=1036.533,304.459,379.798,171.601,43.605,158.401
C08179=1036.525,304.211,379.832,171.596,43.604,158.400
C08180=1036.518,303.963,379.865,171.592,43.602,158.399
C08181=1036.512,303.716,379.899,171.587,43.601,158.399
C08182=1036.505,303.468,379.932,171.584,43.600,158.398
C08183=1036.498,303.221,379.965,171.580,43.598,158.397
C08184=1036.491,302.973,379.998,171.575,43.597,158.397
C08185=1036.484,302.725,380.030,171.571,43.596,158.396
C08186=1036.477,302.477,380.064,171.568,43.595,158.396
C08187=1036.470,302.230,380.096,171.563,43.593,158.395
C08188=1036.463,301.982,380.129,171.559,43.592,158.394
C08189=1036.457,301.735,380.163,171.555,43.590,158.394
C08190=1036.450,301.487,380.196,171.551,43.589,158.393
C08191=1036.444,301.239,380.229,171.547,43.587,158.392
C08192=1036.436,300.992,380.262,171.543,43.586,158.392
C08193=1036.429,300.744,380.295,171.538,43.585,158.391
C08194=1036.422,300.496,380.328,171.534,43.584,158.390
C08195=1036.416,300.248,380.361,171.531,43.582,158.390
C08196=1036.408,300.001,380.394,171.526,43.581,158.389
C08197=1036.402,299.753,380.427,171.522,43.579,158.388
C08198=1036.395,299.505,380.460,171.518,43.578,158.388
C08199=1036.389,299.257,380.492,171.515,43.577,158.387
C08200=1036.382,299.010,380.525,171.510,43.576,158.387
C08201=1036.374,298.762,380.558,171.506,43.574,158.386
C08202=1036.368,298.515,380.591,171.502,43.573,158.385
C08203=1036.361,298.266,380.624,171.499,43.571,158.385
C08204=1036.354,298.019,380.656,171.494,43.570,158.384
C08205=1036.348,297.772,380.689,171.490,43.569,158.384
C08206=1036.341,297.523,380.722,171.486,43.568,158.383
C08207=1036.335,297.276,380.755,171.483,43.567,158.382
C08208=1036.328,297.028,380.787,171.478,43.565,158.382
C08209=1036.321,296.780,380.820,171.474,43.564,158.381
C08210=1036.315,296.532,380.853,171.470,43.562,158.380
C08211=1036.308,296.285,380.886,171.467,43.561,158.380
C08212=1036.301,296.037,380.918,171.462,43.560,158.379
C08213=1036.294,295.789,380.951,171.458,43.559,158.379
C08214=1036.288,295.542,380.984,171.455,43.557,158.378
C08215=1036.280,295.294,381.016,171.451,43.556,158.377
C08216=1036.274,295.046,381.049,171.447,43.555,158.377
C08217=1036.268,294.799,381.082,171.442,43.554,158.376
C08218=1036.260,294.551,381.114,171.439,43.552,158.376
C08219=1036.253,294.303,381.146,171.435,43.551,158.375
C08220=1036.247,294.055,381.178,171.431,43.550,158.374
C08221=1036.240,293.807,381.211,171.427,43.549,158.374
C08222=1036.233,293.559,381.244,171.423,43.548,158.373
C08223=1036.226,293.312,381.276,171.419,43.547,158.373
C08224=1036.220,293.064,381.308,171.416,43.546,158.372
C08225=1036.213,292.816,381.340,171.412,43.544,158.372
C08226=1036.206,292.569,381.373,171.407,43.543,158.371
C08227=1036.199,292.321,381.404,171.404,43.542,158.370
C08228=1036.189,291.970,381.450,171.399,43.540,158.369
C08229=1036.180,291.619,381.495,171.393,43.539,158.369
C08230=1036.170,291.269,381.541,171.388,43.537,158.368
C08231=1036.161,290.918,381.586,171.382,43.535,158.367
C08232=1036.153,290.670,381.619,171.378,43.535,158.367
C08233=1036.146,290.422,381.650,171.375,43.533,158.366
C08234=1036.140,290.175,381.683,171.371,43.532,158.365
C08235=1036.133,289.927,381.714,171.366,43.531,158.365
C08236=1036.126,289.679,381.747,171.363,43.530,158.364
C08237=1036.119,289.431,381.778,171.359,43.529,158.364
C08238=1036.113,289.183,381.811,171.355,43.528,158.363
C08239=1036.106,288.935,381.842,171.352,43.527,158.363
C08240=1036.099,288.688,381.875,171.348,43.526,158.362
C08241=1036.092,288.440,381.906,171.344,43.525,158.362
C08242=1036.085,288.192,381.938,171.340,43.524,158.361
C08243=1036.079,287.944,381.971,171.336,43.523,158.361
C08244=1036.072,287.696,382.002,171.333,43.522,158.360
C08245=1036.065,287.449,382.034,171.329,43.520,158.359
C08246=1036.058,287.201,382.066,171.325,43.520,158.359
C08247=1036.051,286.953,382.097,171.322,43.518,158.358
C08248=1036.045,286.705,382.129,171.317,43.517,158.358
C08249=1036.038,286.457,382.162,171.314,43.517,158.357
C08250=1036.031,286.209,382.193,171.310,43.515,158.357
C08251=1036.024,285.961,382.224,171.306,43.515,158.356
C08252=1036.018,285.713,382.256,171.303,43.513,158.356
C08253=1036.011,285.466,382.288,171.299,43.513,158.355
C08254=1036.004,285.218,382.319,171.295,43.511,158.355
C08255=1035.997,284.970,382.351,171.292,43.511,158.354
C08256=1035.990,284.721,382.383,171.287,43.510,158.354
C08257=1035.983,284.474,382.414,171.284,43.509,158.353
C08258=1035.976,284.226,382.446,171.280,43.508,158.353
C08259=1035.969,283.978,382.476,171.277,43.507,158.352
C08260=1035.962,283.730,382.508,171.273,43.506,158.351
C08261=1035.955,283.482,382.539,171.269,43.505,158.351
C08262=1035.948,283.235,382.571,171.266,43.504,158.350
C08263=1035.942,282.987,382.603,171.262,43.503,158.350
C08264=1035.935,282.739,382.634,171.259,43.502,158.349
C08265=1035.928,282.491,382.666,171.255,43.501,158.349
C08266=1035.921,282.243,382.697,171.251,43.500,158.348
C08267=1035.915,281.995,382.729,171.248,43.499,158.348
C08268=1035.908,281.748,382.760,171.243,43.498,158.347
C08269=1035.901,281.500,382.791,171.240,43.497,158.347
C08270=1035.895,281.252,382.823,171.236,43.496,158.346
C08271=1035.888,281.003,382.854,171.233,43.495,158.346
C08272=1035.881,280.755,382.885,171.229,43.494,158.345
C08273=1035.875,280.507,382.916,171.225,43.493,158.345
C08274=1035.868,280.260,382.948,171.222,43.492,158.344
C08275=1035.861,280.012,382.979,171.218,43.491,158.344
C08276=1035.854,279.764,383.011,171.215,43.491,158.343
C08277=1035.848,279.516,383.042,171.211,43.489,158.343
C08278=1035.841,279.268,383.074,171.208,43.489,158.342
C08279=1035.834,279.020,383.105,171.204,43.487,158.342
C08280=1035.828,278.772,383.136,171.200,43.487,158.341
C08281=1035.821,278.524,383.167,171.197,43.486,158.341
C08282=1035.814,278.276,383.198,171.193,43.485,158.340
C08283=1035.808,278.029,383.229,171.190,43.484,158.340
C08284=1035.798,277.689,383.271,171.185,43.483,158.339
C08285=1035.789,277.351,383.314,171.180,43.482,158.339
C08286=1035.780,277.012,383.356,171.175,43.480,158.338
C08287=1035.770,276.673,383.398,171.171,43.479,158.337
C08288=1035.764,276.426,383.430,171.167,43.478,158.337
C08289=1035.757,276.177,383.460,171.164,43.478,158.336
C08290=1035.750,275.929,383.491,171.160,43.477,158.336
C08291=1035.743,275.682,383.523,171.157,43.476,158.335
C08292=1035.737,275.434,383.553,171.153,43.475,158.335
C08293=1035.730,275.186,383.584,171.150,43.474,158.334
C08294=1035.723,274.938,383.615,171.146,43.474,158.334
C08295=1035.717,274.690,383.646,171.142,43.472,158.333
C08296=1035.710,274.441,383.677,171.139,43.472,158.333
C08297=1035.703,274.194,383.707,171.135,43.471,158.333
C08298=1035.697,273.946,383.738,171.132,43.470,158.332
C08299=1035.689,273.698,383.769,171.128,43.469,158.332
C08300=1035.683,273.450,383.799,171.125,43.468,158.331
C08301=1035.676,273.202,383.831,171.121,43.468,158.331
C08302=1035.669,272.954,383.861,171.118,43.467,158.330
C08303=1035.662,272.706,383.892,171.114,43.466,158.330
C08304=1035.657,272.458,383.923,171.111,43.466,158.329
C08305=1035.649,272.210,383.953,171.107,43.464,158.329
C08306=1035.643,271.962,383.984,171.104,43.464,158.328
C08307=1035.636,271.714,384.014,171.100,43.463,158.328
C08308=1035.629,271.466,384.046,171.097,43.462,158.328
C08309=1035.623,271.218,384.076,171.093,43.462,158.327
C08310=1035.616,270.970,384.106,171.090,43.461,158.327
C08311=1035.609,270.721,384.137,171.086,43.460,158.326
C08312=1035.602,270.473,384.168,171.084,43.459,158.326
C08313=1035.596,270.226,384.198,171.080,43.458,158.325
C08314=1035.589,269.977,384.228,171.077,43.457,158.325
C08315=1035.582,269.729,384.258,171.073,43.457,158.324
C08316=1035.575,269.481,384.290,171.070,43.456,158.324
C08317=1035.569,269.234,384.320,171.066,43.455,158.324
C08318=1035.562,268.985,384.350,171.063,43.455,158.323
C08319=1035.555,268.737,384.380,171.059,43.454,158.323
C08320=1035.549,268.489,384.411,171.056,43.453,158.322
C08321=1035.542,268.242,384.442,171.052,43.453,158.322
C08322=1035.535,267.993,384.472,171.049,43.452,158.321
C08323=1035.528,267.745,384.503,171.046,43.451,158.321
C08324=1035.522,267.497,384.532,171.043,43.450,158.321
C08325=1035.515,267.249,384.563,171.040,43.450,158.320
C08326=1035.508,267.001,384.593,171.036,43.449,158.320
C08327=1035.502,266.753,384.623,171.033,43.448,158.319
C08328=1035.495,266.505,384.654,171.029,43.448,158.319
C08329=1035.488,266.256,384.684,171.026,43.447,158.318
C08330=1035.481,266.009,384.713,171.022,43.446,158.318
C08331=1035.475,265.760,384.744,171.019,43.445,158.318
C08332=1035.468,265.512,384.774,171.016,43.445,158.317
C08333=1035.461,265.265,384.804,171.013,43.444,158.317
C08334=1035.455,265.016,384.835,171.009,43.443,158.316
C08335=1035.448,264.768,384.865,171.006,43.442,158.316
C08336=1035.441,264.520,384.895,171.002,43.442,158.315
C08337=1035.434,264.272,384.925,170.999,43.441,158.315
C08338=1035.427,264.024,384.955,170.995,43.440,158.315
C08339=1035.421,263.776,384.985,170.993,43.440,158.314
C08340=1035.412,263.442,385.026,170.988,43.439,158.314
C08341=1035.403,263.108,385.066,170.984,43.438,158.313
C08342=1035.394,262.774,385.107,170.979,43.437,158.313
C08343=1035.385,262.440,385.147,170.975,43.436,158.312
C08344=1035.378,262.191,385.177,170.971,43.436,158.312
C08345=1035.372,261.944,385.207,170.969,43.435,158.311
C08346=1035.365,261.695,385.236,170.965,43.434,158.311
C08347=1035.358,261.447,385.266,170.962,43.434,158.310
C08348=1035.351,261.199,385.296,170.958,43.433,158.310
C08349=1035.344,260.950,385.326,170.955,43.433,158.310
C08350=1035.338,260.703,385.355,170.951,43.432,158.309
C08351=1035.330,260.455,385.386,170.949,43.432,158.309
C08352=1035.324,260.207,385.415,170.946,43.431,158.308
C08353=1035.317,259.958,385.445,170.942,43.430,158.308
C08354=1035.310,259.710,385.474,170.939,43.430,158.308
C08355=1035.303,259.462,385.503,170.936,43.429,158.307
C08356=1035.296,259.214,385.533,170.932,43.429,158.307
C08357=1035.290,258.966,385.562,170.930,43.429,158.307
C08358=1035.282,258.718,385.593,170.926,43.428,158.306
C08359=1035.276,258.469,385.622,170.923,43.427,158.306
C08360=1035.269,258.221,385.652,170.919,43.426,158.305
C08361=1035.262,257.973,385.681,170.916,43.426,158.305
C08362=1035.256,257.725,385.711,170.913,43.426,158.305
C08363=1035.249,257.476,385.740,170.910,43.425,158.304
C08364=1035.241,257.229,385.769,170.907,43.425,158.304
C08365=1035.235,256.980,385.799,170.903,43.424,158.304
C08366=1035.228,256.732,385.828,170.900,43.423,158.303
C08367=1035.221,256.484,385.858,170.897,43.423,158.303
C08368=1035.215,256.236,385.887,170.894,43.422,158.302
C08369=1035.208,255.988,385.917,170.891,43.422,158.302
C08370=1035.202,255.739,385.946,170.888,43.422,158.302
C08371=1035.194,255.491,385.976,170.884,43.421,158.301
C08372=1035.187,255.243,386.005,170.882,43.420,158.301
C08373=1035.181,254.995,386.034,170.878,43.420,158.301
C08374=1035.174,254.747,386.064,170.875,43.419,158.300
C08375=1035.167,254.498,386.093,170.871,43.419,158.300
C08376=1035.161,254.250,386.122,170.869,43.418,158.300
C08377=1035.154,254.003,386.152,170.866,43.418,158.299
C08378=1035.147,253.754,386.182,170.862,43.417,158.299
C08379=1035.140,253.506,386.210,170.859,43.417,158.298
C08380=1035.133,253.258,386.240,170.857,43.416,158.298
C08381=1035.127,253.010,386.269,170.853,43.415,158.298
C08382=1035.121,252.761,386.298,170.850,43.415,158.297
C08383=1035.114,252.513,386.328,170.846,43.414,158.297
C08384=1035.107,252.265,386.357,170.844,43.414,158.297
C08385=1035.100,252.017,386.386,170.841,43.414,158.296
C08386=1035.094,251.768,386.415,170.837,43.413,158.296
C08387=1035.087,251.520,386.444,170.834,43.413,158.295
C08388=1035.080,251.271,386.474,170.831,43.412,158.295
C08389=1035.074,251.024,386.503,170.828,43.411,158.295
C08390=1035.068,250.776,386.532,170.825,43.411,158.294
C08391=1035.061,250.527,386.562,170.822,43.410,158.294
C08392=1035.054,250.279,386.590,170.819,43.410,158.294
C08393=1035.048,250.031,386.619,170.815,43.409,158.293
C08394=1035.041,249.782,386.649,170.813,43.409,158.293
C08395=1035.034,249.535,386.679,170.810,43.408,158.293
C08396=1035.025,249.199,386.718,170.805,43.408,158.292
C08397=1035.016,248.863,386.756,170.802,43.407,158.292
C08398=1035.007,248.528,386.796,170.797,43.406,158.291
C08399=1034.999,248.193,386.835,170.794,43.405,158.291
C08400=1034.993,247.944,386.865,170.790,43.405,158.290
C08401=1034.985,247.696,386.893,170.787,43.405,158.290
C08402=1034.979,247.448,386.922,170.784,43.404,158.290
C08403=1034.972,247.200,386.951,170.781,43.404,158.289
C08404=1034.966,246.951,386.980,170.778,43.403,158.289
C08405=1034.959,246.703,387.010,170.775,43.403,158.289
C08406=1034.953,246.455,387.039,170.772,43.402,158.288
C08407=1034.946,246.207,387.067,170.769,43.401,158.288
C08408=1034.940,245.959,387.096,170.766,43.401,158.288
C08409=1034.934,245.710,387.125,170.763,43.400,158.287
C08410=1034.927,245.462,387.155,170.761,43.400,158.287
C08411=1034.921,245.213,387.184,170.757,43.399,158.286
C08412=1034.914,244.966,387.212,170.754,43.399,158.286
C08413=1034.907,244.718,387.241,170.751,43.398,158.286
C08414=1034.901,244.469,387.270,170.748,43.398,158.285
C08415=1034.893,244.221,387.299,170.745,43.398,158.285
C08416=1034.887,243.973,387.328,170.742,43.397,158.285
C08417=1034.881,243.724,387.356,170.739,43.397,158.284
C08418=1034.874,243.476,387.385,170.737,43.396,158.284
C08419=1034.867,243.228,387.414,170.733,43.396,158.284
C08420=1034.860,242.980,387.443,170.730,43.396,158.283
C08421=1034.855,242.731,387.471,170.728,43.395,158.283
C08422=1034.848,242.483,387.500,170.724,43.395,158.283
C08423=1034.841,242.235,387.529,170.721,43.394,158.282
C08424=1034.834,241.986,387.557,170.719,43.394,158.282
C08425=1034.828,241.738,387.586,170.715,43.393,158.282
C08426=1034.821,241.490,387.614,170.713,43.393,158.281
C08427=1034.815,241.242,387.643,170.710,43.393,158.281
C08428=1034.808,240.993,387.671,170.706,43.392,158.281
C08429=1034.802,240.745,387.700,170.704,43.392,158.280
C08430=1034.795,240.497,387.729,170.700,43.391,158.280
C08431=1034.788,240.248,387.757,170.698,43.391,158.280
C08432=1034.781,240.000,387.786,170.695,43.391,158.280
C08433=1034.774,239.752,387.814,170.691,43.390,158.279
C08434=1034.768,239.503,387.842,170.689,43.390,158.279
C08435=1034.761,239.256,387.871,170.686,43.390,158.279
C08436=1034.754,239.006,387.899,170.683,43.389,158.278
C08437=1034.747,238.759,387.927,170.680,43.389,158.278
C08438=1034.741,238.510,387.956,170.677,43.389,158.278
C08439=1034.734,238.262,387.984,170.674,43.388,158.277
C08440=1034.727,238.014,388.012,170.671,43.388,158.277
C08441=1034.721,237.765,388.041,170.669,43.387,158.277
C08442=1034.714,237.517,388.069,170.666,43.387,158.276
C08443=1034.707,237.269,388.097,170.663,43.386,158.276
C08444=1034.700,237.020,388.125,170.660,43.386,158.276
C08445=1034.694,236.771,388.154,170.657,43.386,158.276
C08446=1034.687,236.523,388.182,170.654,43.385,158.275
C08447=1034.680,236.275,388.210,170.651,43.385,158.275
C08448=1034.673,236.027,388.238,170.649,43.385,158.275
C08449=1034.668,235.778,388.267,170.646,43.385,158.274
C08450=1034.661,235.530,388.294,170.643,43.384,158.274
C08451=1034.654,235.282,388.323,170.640,43.384,158.274
C08452=1034.645,234.940,388.361,170.636,43.383,158.273
C08453=1034.636,234.599,388.399,170.632,43.383,158.273
C08454=1034.626,234.258,388.439,170.629,43.383,158.272
C08455=1034.617,233.916,388.477,170.624,43.382,158.272
C08456=1034.610,233.668,388.505,170.622,43.382,158.272
C08457=1034.604,233.419,388.533,170.618,43.381,158.271
C08458=1034.597,233.172,388.561,170.616,43.381,158.271
C08459=1034.591,232.923,388.590,170.613,43.381,158.271
C08460=1034.584,232.674,388.617,170.611,43.380,158.271
C08461=1034.577,232.427,388.646,170.607,43.380,158.270
C08462=1034.570,232.178,388.674,170.605,43.379,158.270
C08463=1034.564,231.929,388.702,170.602,43.379,158.270
C08464=1034.558,231.681,388.730,170.599,43.379,158.269
C08465=1034.551,231.433,388.757,170.596,43.378,158.269
C08466=1034.544,231.185,388.786,170.593,43.378,158.269
C08467=1034.537,230.936,388.813,170.591,43.378,158.268
C08468=1034.531,230.688,388.841,170.587,43.378,158.268
C08469=1034.524,230.439,388.869,170.585,43.378,158.268
C08470=1034.517,230.191,388.897,170.582,43.377,158.268
C08471=1034.511,229.942,388.924,170.579,43.377,158.267
C08472=1034.504,229.694,388.952,170.576,43.377,158.267
C08473=1034.498,229.446,388.980,170.574,43.376,158.267
C08474=1034.491,229.198,389.007,170.572,43.376,158.267
C08475=1034.484,228.950,389.036,170.568,43.375,158.266
C08476=1034.478,228.701,389.064,170.566,43.375,158.266
C08477=1034.472,228.453,389.092,170.563,43.375,158.266
C08478=1034.465,228.204,389.119,170.560,43.375,158.265
C08479=1034.458,227.956,389.147,170.557,43.375,158.265
C08480=1034.451,227.708,389.174,170.555,43.374,158.265
C08481=1034.444,227.459,389.202,170.552,43.374,158.265
C08482=1034.437,227.211,389.230,170.549,43.373,158.264
C08483=1034.431,226.962,389.257,170.546,43.373,158.264
C08484=1034.424,226.713,389.285,170.544,43.373,158.264
C08485=1034.418,226.465,389.312,170.540,43.373,158.263
C08486=1034.410,226.217,389.339,170.538,43.373,158.263
C08487=1034.404,225.968,389.367,170.535,43.373,158.263
C08488=1034.397,225.720,389.395,170.533,43.372,158.263
C08489=1034.390,225.472,389.423,170.529,43.372,158.262
C08490=1034.383,225.223,389.450,170.527,43.372,158.262
C08491=1034.377,224.975,389.478,170.524,43.372,158.262
C08492=1034.370,224.727,389.504,170.522,43.372,158.262
C08493=1034.364,224.478,389.532,170.518,43.372,158.261
C08494=1034.357,224.230,389.560,170.516,43.371,158.261
C08495=1034.350,223.981,389.587,170.514,43.370,158.261
C08496=1034.344,223.733,389.615,170.510,43.370,158.260
C08497=1034.336,223.484,389.641,170.508,43.370,158.260
C08498=1034.330,223.236,389.669,170.505,43.370,158.260
C08499=1034.324,222.988,389.697,170.503,43.370,158.260
C08500=1034.317,222.740,389.724,170.499,43.370,158.259
C08501=1034.310,222.491,389.752,170.497,43.369,158.259
C08502=1034.303,222.242,389.778,170.495,43.369,158.259
C08503=1034.297,221.994,389.806,170.492,43.369,158.259
C08504=1034.290,221.745,389.834,170.490,43.369,158.258
C08505=1034.284,221.497,389.861,170.486,43.369,158.258
C08506=1034.277,221.249,389.888,170.484,43.368,158.258
C08507=1034.270,221.000,389.915,170.482,43.368,158.258
C08508=1034.261,220.651,389.953,170.477,43.368,158.257
C08509=1034.252,220.303,389.993,170.474,43.368,158.257
C08510=1034.243,219.953,390.031,170.470,43.367,158.256
C08511=1034.233,219.604,390.069,170.466,43.367,158.256
C08512=1034.226,219.356,390.096,170.464,43.367,158.256
C08513=1034.220,219.108,390.123,170.461,43.367,158.256
C08514=1034.213,218.860,390.150,170.459,43.366,158.255
C08515=1034.206,218.611,390.178,170.455,43.366,158.255
C08516=1034.199,218.363,390.204,170.453,43.366,158.255
C08517=1034.192,218.114,390.232,170.451,43.366,158.255
C08518=1034.186,217.866,390.258,170.448,43.366,158.254
C08519=1034.179,217.618,390.285,170.445,43.365,158.254
C08520=1034.172,217.369,390.312,170.442,43.365,158.254
C08521=1034.165,217.120,390.340,170.440,43.365,158.254
C08522=1034.159,216.871,390.367,170.438,43.365,158.253
C08523=1034.152,216.624,390.393,170.434,43.365,158.253
C08524=1034.146,216.375,390.420,170.432,43.364,158.253
C08525=1034.139,216.126,390.447,170.430,43.364,158.253
C08526=1034.132,215.878,390.475,170.427,43.364,158.252
C08527=1034.125,215.630,390.501,170.424,43.364,158.252
C08528=1034.119,215.381,390.528,170.421,43.364,158.252
C08529=1034.112,215.132,390.555,170.419,43.364,158.252
C08530=1034.105,214.885,390.582,170.417,43.364,158.252
C08531=1034.098,214.636,390.609,170.414,43.364,158.251
C08532=1034.092,214.387,390.636,170.411,43.363,158.251
C08533=1034.085,214.139,390.663,170.409,43.363,158.251
C08534=1034.079,213.890,390.689,170.406,43.363,158.251
C08535=1034.072,213.642,390.716,170.404,43.363,158.250
C08536=1034.065,213.393,390.743,170.401,43.362,158.250
C08537=1034.058,213.145,390.770,170.398,43.362,158.250
C08538=1034.052,212.896,390.797,170.396,43.362,158.250
C08539=1034.045,212.648,390.824,170.394,43.362,158.249
C08540=1034.039,212.400,390.850,170.390,43.362,158.249
C08541=1034.032,212.151,390.877,170.388,43.361,158.249
C08542=1034.025,211.902,390.904,170.386,43.361,158.249
C08543=1034.019,211.654,390.931,170.383,43.361,158.248
C08544=1034.012,211.405,390.958,170.380,43.361,158.248
C08545=1034.005,211.157,390.985,170.378,43.361,158.248
C08546=1033.998,210.909,391.011,170.375,43.360,158.248
C08547=1033.992,210.660,391.038,170.373,43.361,158.247
C08548=1033.985,210.411,391.064,170.371,43.361,158.247
C08549=1033.978,210.163,391.090,170.367,43.360,158.247
C08550=1033.972,209.915,391.118,170.365,43.360,158.247
C08551=1033.964,209.666,391.144,170.363,43.360,158.246
C08552=1033.958,209.418,391.170,170.361,43.360,158.246
C08553=1033.952,209.169,391.197,170.357,43.360,158.246
C08554=1033.944,208.920,391.224,170.355,43.359,158.246
C08555=1033.938,208.672,391.250,170.353,43.360,158.246
C08556=1033.932,208.423,391.277,170.350,43.360,158.245
C08557=1033.925,208.175,391.303,170.348,43.359,158.245
C08558=1033.918,207.927,391.330,170.345,43.359,158.245
C08559=1033.911,207.678,391.357,170.342,43.359,158.245
C08560=1033.905,207.430,391.383,170.340,43.359,158.244
C08561=1033.898,207.181,391.410,170.338,43.359,158.244
C08562=1033.891,206.932,391.436,170.336,43.359,158.244
C08563=1033.884,206.684,391.462,170.332,43.359,158.244
C08564=1033.875,206.341,391.499,170.329,43.359,158.243
C08565=1033.865,205.998,391.535,170.326,43.358,158.243
C08566=1033.855,205.655,391.571,170.323,43.358,158.243
C08567=1033.846,205.311,391.607,170.319,43.358,158.243
C08568=1033.821,204.262,391.713,169.988,43.254,158.195
C08569=1033.814,204.013,391.738,169.985,43.254,158.195
C08570=1033.808,203.765,391.763,169.982,43.255,158.194
C08571=1033.802,203.515,391.788,169.978,43.255,158.194
C08572=1033.797,203.267,391.813,169.975,43.256,158.194
C08573=1033.790,203.019,391.838,169.971,43.257,158.194
C08574=1033.784,202.770,391.864,169.968,43.257,158.194
C08575=1033.778,202.521,391.888,169.964,43.259,158.194
C08576=1033.772,202.272,391.914,169.961,43.259,158.194
C08577=1033.766,202.024,391.938,169.958,43.260,158.194
C08578=1033.760,201.775,391.963,169.954,43.260,158.193
C08579=1033.754,201.527,391.988,169.950,43.261,158.193
C08580=1033.747,201.278,392.013,169.947,43.261,158.193
C08581=1033.742,201.029,392.038,169.943,43.262,158.193
C08582=1033.736,200.781,392.063,169.940,43.263,158.193
C08583=1033.730,200.531,392.088,169.936,43.263,158.193
C08584=1033.723,200.283,392.112,169.933,43.265,158.193
C08585=1033.717,200.034,392.137,169.930,43.265,158.193
C08586=1033.711,199.786,392.161,169.926,43.266,158.192
C08587=1033.705,199.537,392.186,169.924,43.267,158.192
C08588=1033.698,199.288,392.211,169.920,43.268,158.192
C08589=1033.692,199.039,392.235,169.916,43.268,158.192
C08590=1033.685,198.791,392.260,169.913,43.269,158.192
C08591=1033.680,198.542,392.284,169.910,43.270,158.192
C08592=1033.673,198.293,392.308,169.907,43.271,158.192
C08593=1033.667,198.044,392.334,169.902,43.271,158.192
C08594=1033.660,197.795,392.358,169.900,43.272,158.192
C08595=1033.655,197.547,392.382,169.897,43.273,158.191
C08596=1033.648,197.299,392.407,169.893,43.274,158.191
C08597=1033.642,197.049,392.431,169.890,43.275,158.191
C08598=1033.637,196.801,392.456,169.886,43.276,158.191
C08599=1033.630,196.552,392.480,169.883,43.276,158.191
C08600=1033.624,196.303,392.505,169.880,43.277,158.191
C08601=1033.618,196.055,392.529,169.876,43.278,158.191
C08602=1033.612,195.806,392.554,169.873,43.279,158.191
C08603=1033.605,195.557,392.578,169.870,43.280,158.191
C08604=1033.600,195.308,392.602,169.866,43.280,158.191
C08605=1033.593,195.060,392.627,169.863,43.282,158.191
C08606=1033.587,194.811,392.652,169.860,43.282,158.190
C08607=1033.581,194.563,392.675,169.856,43.283,158.190
C08608=1033.575,194.313,392.700,169.853,43.284,158.190
C08609=1033.568,194.065,392.725,169.850,43.285,158.190
C08610=1033.563,193.816,392.749,169.846,43.285,158.190
C08611=1033.556,193.567,392.773,169.843,43.286,158.190
C08612=1033.550,193.318,392.798,169.840,43.287,158.190
C08613=1033.544,193.070,392.821,169.836,43.288,158.190
C08614=1033.538,192.820,392.846,169.833,43.289,158.190
C08615=1033.532,192.573,392.870,169.830,43.289,158.190
C08616=1033.525,192.324,392.894,169.826,43.291,158.190
C08617=1033.520,192.075,392.919,169.823,43.291,158.189
C08618=1033.514,191.826,392.943,169.821,43.292,158.189
C08619=1033.508,191.577,392.967,169.817,43.293,158.189
C08620=1033.502,191.329,392.991,169.813,43.294,158.189
C08621=1033.496,191.079,393.015,169.811,43.295,158.189
C08622=1033.490,190.831,393.039,169.808,43.295,158.189
C08623=1033.483,190.583,393.064,169.804,43.297,158.189
C08624=1033.477,190.334,393.088,169.801,43.297,158.189
C08625=1033.471,190.085,393.113,169.798,43.298,158.189
C08626=1033.465,189.837,393.136,169.795,43.299,158.189
C08627=1033.460,189.587,393.161,169.791,43.300,158.189
C08628=1033.454,189.339,393.185,169.788,43.301,158.189
C08629=1033.446,189.054,393.212,169.784,43.302,158.188
C08630=1033.440,188.771,393.240,169.781,43.303,158.188
C08631=1033.433,188.487,393.267,169.777,43.304,158.188
C08632=1033.426,188.203,393.294,169.773,43.305,158.188
C08633=1033.420,187.954,393.318,169.770,43.305,158.188
C08634=1033.415,187.706,393.343,169.767,43.307,158.188
C08635=1033.408,187.457,393.367,169.764,43.307,158.188
C08636=1033.403,187.208,393.391,169.760,43.308,158.188
C08637=1033.397,186.960,393.415,169.757,43.309,158.188
C08638=1033.391,186.710,393.439,169.755,43.310,158.188
C08639=1033.385,186.462,393.463,169.751,43.311,158.188
C08640=1033.379,186.213,393.488,169.749,43.312,158.188
C08641=1033.373,185.965,393.511,169.745,43.313,158.188
C08642=1033.367,185.715,393.536,169.742,43.313,158.187
C08643=1033.361,185.466,393.559,169.739,43.314,158.187
C08644=1033.355,185.218,393.582,169.736,43.315,158.187
C08645=1033.349,184.969,393.607,169.733,43.316,158.187
C08646=1033.343,184.721,393.631,169.729,43.317,158.187
C08647=1033.337,184.471,393.655,169.726,43.318,158.187
C08648=1033.331,184.223,393.679,169.723,43.318,158.187
C08649=1033.326,183.974,393.703,169.720,43.320,158.187
C08650=1033.320,183.725,393.727,169.717,43.320,158.187
C08651=1033.313,183.476,393.750,169.714,43.321,158.187
C08652=1033.308,183.228,393.775,169.710,43.322,158.187
C08653=1033.302,182.978,393.798,169.707,43.323,158.187
C08654=1033.296,182.730,393.821,169.705,43.324,158.187
C08655=1033.289,182.481,393.846,169.702,43.326,158.187
C08656=1033.283,182.232,393.868,169.698,43.326,158.187
C08657=1033.276,181.983,393.892,169.695,43.327,158.187
C08658=1033.270,181.735,393.915,169.692,43.329,158.187
C08659=1033.264,181.486,393.938,169.689,43.330,158.187
C08660=1033.258,181.237,393.962,169.686,43.331,158.187
C08661=1033.252,180.988,393.985,169.682,43.332,158.186
C08662=1033.246,180.739,394.009,169.679,43.333,158.186
C08663=1033.240,180.491,394.032,169.677,43.334,158.187
C08664=1033.233,180.242,394.055,169.674,43.335,158.187
C08665=1033.226,179.993,394.079,169.670,43.337,158.186
C08666=1033.221,179.744,394.102,169.667,43.338,158.187
C08667=1033.214,179.495,394.126,169.664,43.338,158.186
C08668=1033.208,179.246,394.149,169.661,43.340,158.186
C08669=1033.202,178.998,394.172,169.658,43.341,158.186
C08670=1033.196,178.748,394.196,169.655,43.342,158.186
C08671=1033.190,178.500,394.218,169.652,43.343,158.186
C08672=1033.183,178.251,394.242,169.649,43.344,158.186
C08673=1033.177,178.002,394.265,169.646,43.345,158.186
C08674=1033.171,177.754,394.289,169.643,43.346,158.186
C08675=1033.165,177.505,394.312,169.639,43.348,158.186
C08676=1033.159,177.255,394.335,169.636,43.349,158.186
C08677=1033.152,177.007,394.358,169.634,43.350,158.186
C08678=1033.147,176.758,394.381,169.631,43.351,158.186
C08679=1033.140,176.509,394.404,169.628,43.352,158.186
C08680=1033.134,176.260,394.428,169.624,43.353,158.186
C08681=1033.128,176.011,394.451,169.621,43.354,158.186
C08682=1033.122,175.763,394.473,169.618,43.355,158.186
C08683=1033.115,175.514,394.497,169.615,43.357,158.186
C08684=1033.110,175.265,394.520,169.613,43.358,158.186
C08685=1033.104,175.016,394.543,169.610,43.359,158.186
C08686=1033.098,174.767,394.566,169.607,43.360,158.186
C08687=1033.092,174.518,394.590,169.603,43.361,158.186
C08688=1033.085,174.270,394.612,169.600,43.362,158.186
C08689=1033.079,174.021,394.635,169.597,43.363,158.186
C08690=1033.074,173.772,394.658,169.594,43.364,158.186
C08691=1033.067,173.523,394.682,169.592,43.365,158.186
C08692=1033.061,173.274,394.705,169.589,43.367,158.186
C08693=1033.054,172.990,394.731,169.585,43.368,158.186
C08694=1033.047,172.706,394.757,169.582,43.369,158.186
C08695=1033.041,172.422,394.784,169.578,43.371,158.186
C08696=1033.034,172.137,394.810,169.575,43.372,158.186
C08697=1033.027,171.888,394.833,169.572,43.373,158.186
C08698=1033.021,171.639,394.856,169.568,43.374,158.186
C08699=1033.015,171.391,394.879,169.566,43.375,158.186
C08700=1033.009,171.142,394.902,169.563,43.376,158.186
C08701=1033.004,170.893,394.925,169.560,43.377,158.186
C08702=1032.998,170.644,394.948,169.557,43.378,158.186
C08703=1032.991,170.395,394.971,169.554,43.380,158.186
C08704=1032.985,170.146,394.994,169.552,43.381,158.186
C08705=1032.979,169.897,395.017,169.549,43.382,158.186
C08706=1032.974,169.648,395.040,169.546,43.383,158.186
C08707=1032.968,169.399,395.063,169.543,43.384,158.186
C08708=1032.961,169.151,395.086,169.539,43.385,158.186
C08709=1032.955,168.902,395.109,169.536,43.386,158.186
C08710=1032.950,168.653,395.132,169.533,43.387,158.186
C08711=1032.943,168.404,395.155,169.530,43.389,158.186
C08712=1032.937,168.155,395.177,169.528,43.390,158.186
C08713=1032.931,167.906,395.200,169.525,43.391,158.186
C08714=1032.925,167.657,395.223,169.522,43.392,158.186
C08715=1032.920,167.408,395.246,169.519,43.393,158.186
C08716=1032.914,167.160,395.269,169.516,43.395,158.186
C08717=1032.907,166.911,395.292,169.513,43.395,158.186
C08718=1032.902,166.662,395.314,169.510,43.396,158.186
C08719=1032.896,166.413,395.337,169.508,43.397,158.186
C08720=1032.890,166.164,395.360,169.505,43.399,158.186
C08721=1032.884,165.916,395.383,169.502,43.400,158.186
C08722=1032.878,165.666,395.405,169.499,43.401,158.186
C08723=1032.873,165.417,395.428,169.496,43.402,158.186
C08724=1032.867,165.168,395.451,169.494,43.403,158.186
C08725=1032.861,164.920,395.474,169.491,43.405,158.186
C08726=1032.855,164.671,395.496,169.488,43.406,158.186
C08727=1032.849,164.422,395.519,169.485,43.407,158.186
C08728=1032.843,164.173,395.542,169.482,43.407,158.186
C08729=1032.837,163.924,395.565,169.479,43.409,158.186
C08730=1032.831,163.676,395.587,169.476,43.410,158.186
C08731=1032.826,163.426,395.610,169.473,43.411,158.186
C08732=1032.820,163.177,395.632,169.471,43.412,158.186
C08733=1032.814,162.928,395.655,169.468,43.413,158.186
C08734=1032.808,162.680,395.678,169.465,43.415,158.186
C08735=1032.802,162.431,395.701,169.462,43.416,158.186
C08736=1032.796,162.182,395.724,169.459,43.417,158.186
C08737=1032.791,161.932,395.746,169.457,43.418,158.186
C08738=1032.784,161.684,395.768,169.454,43.419,158.186
C08739=1032.779,161.435,395.791,169.451,43.420,158.186
C08740=1032.773,161.186,395.814,169.448,43.421,158.186
C08741=1032.767,160.937,395.837,169.445,43.422,158.186
C08742=1032.761,160.688,395.859,169.442,43.423,158.186
C08743=1032.755,160.439,395.882,169.439,43.425,158.186
C08744=1032.749,160.190,395.905,169.437,43.426,158.186
C08745=1032.743,159.942,395.927,169.434,43.427,158.186
C08746=1032.738,159.692,395.949,169.431,43.428,158.186
C08747=1032.731,159.443,395.972,169.428,43.429,158.186
C08748=1032.726,159.194,395.994,169.425,43.431,158.186
C08749=1032.719,158.945,396.016,169.422,43.432,158.186
C08750=1032.714,158.697,396.037,169.420,43.434,158.186
C08751=1032.708,158.448,396.060,169.417,43.435,158.186
C08752=1032.701,158.199,396.083,169.414,43.436,158.186
C08753=1032.695,157.950,396.104,169.411,43.437,158.186
C08754=1032.690,157.701,396.127,169.408,43.438,158.186
C08755=1032.683,157.452,396.149,169.406,43.440,158.186
C08756=1032.677,157.204,396.171,169.403,43.441,158.186
C08757=1032.670,156.918,396.196,169.400,43.443,158.186
C08758=1032.663,156.634,396.222,169.396,43.444,158.186
C08759=1032.657,156.349,396.247,169.394,43.445,158.186
C08760=1032.650,156.064,396.273,169.391,43.447,158.186
C08761=1032.644,155.815,396.294,169.388,43.448,158.186
C08762=1032.637,155.567,396.317,169.385,43.449,158.186
C08763=1032.632,155.317,396.339,169.382,43.451,158.186
C08764=1032.625,155.069,396.361,169.380,43.452,158.186
C08765=1032.619,154.819,396.383,169.377,43.453,158.186
C08766=1032.614,154.570,396.406,169.374,43.455,158.186
C08767=1032.607,154.321,396.427,169.371,43.456,158.186
C08768=1032.601,154.072,396.449,169.368,43.457,158.186
C08769=1032.595,153.824,396.471,169.366,43.458,158.186
C08770=1032.590,153.575,396.493,169.363,43.460,158.187
C08771=1032.583,153.326,396.516,169.360,43.461,158.187
C08772=1032.577,153.077,396.537,169.357,43.463,158.187
C08773=1032.571,152.828,396.559,169.355,43.464,158.187
C08774=1032.565,152.578,396.580,169.352,43.465,158.187
C08775=1032.558,152.330,396.603,169.349,43.466,158.187
C08776=1032.554,152.081,396.625,169.346,43.468,158.187
C08777=1032.548,151.832,396.646,169.343,43.469,158.187
C08778=1032.541,151.583,396.669,169.341,43.470,158.187
C08779=1032.535,151.334,396.690,169.338,43.472,158.187
C08780=1032.529,151.085,396.712,169.335,43.473,158.187
C08781=1032.523,150.836,396.734,169.332,43.475,158.187
C08782=1032.517,150.588,396.756,169.331,43.476,158.187
C08783=1032.511,150.338,396.778,169.328,43.477,158.187
C08784=1032.505,150.089,396.799,169.325,43.478,158.187
C08785=1032.499,149.840,396.821,169.322,43.480,158.187
C08786=1032.492,149.591,396.843,169.319,43.481,158.187
C08787=1032.487,149.343,396.865,169.317,43.482,158.187
C08788=1032.481,149.094,396.886,169.314,43.483,158.187
C08789=1032.475,148.844,396.908,169.311,43.485,158.187
C08790=1032.468,148.595,396.930,169.308,43.486,158.187
C08791=1032.463,148.346,396.952,169.306,43.488,158.187
C08792=1032.457,148.098,396.974,169.303,43.489,158.187
C08793=1032.451,147.848,396.995,169.300,43.491,158.188
C08794=1032.445,147.599,397.017,169.297,43.492,158.188
C08795=1032.439,147.350,397.039,169.295,43.493,158.188
C08796=1032.433,147.102,397.060,169.293,43.494,158.188
C08797=1032.427,146.852,397.082,169.290,43.496,158.188
C08798=1032.421,146.603,397.103,169.287,43.497,158.188
C08799=1032.415,146.354,397.125,169.284,43.498,158.188
C08800=1032.408,146.105,397.147,169.282,43.500,158.188
C08801=1032.403,145.856,397.168,169.279,43.501,158.188
C08802=1032.397,145.607,397.189,169.276,43.503,158.188
C08803=1032.390,145.358,397.210,169.273,43.504,158.188
C08804=1032.384,145.109,397.232,169.271,43.506,158.188
C08805=1032.378,144.860,397.253,169.268,43.507,158.188
C08806=1032.372,144.611,397.275,169.265,43.509,158.188
C08807=1032.366,144.362,397.297,169.262,43.510,158.188
C08808=1032.360,144.113,397.318,169.261,43.511,158.188
C08809=1032.354,143.864,397.340,169.258,43.513,158.189
C08810=1032.348,143.615,397.361,169.255,43.514,158.189
C08811=1032.341,143.366,397.382,169.252,43.516,158.189
C08812=1032.335,143.118,397.403,169.250,43.517,158.189
C08813=1032.329,142.869,397.425,169.247,43.518,158.189
C08814=1032.323,142.619,397.447,169.244,43.520,158.189
C08815=1032.317,142.371,397.468,169.241,43.521,158.189
C08816=1032.312,142.121,397.489,169.239,43.522,158.189
C08817=1032.305,141.872,397.511,169.237,43.524,158.189
C08818=1032.299,141.623,397.532,169.234,43.525,158.189
C08819=1032.293,141.374,397.553,169.231,43.526,158.189
C08820=1032.287,141.125,397.575,169.229,43.528,158.189
C08821=1032.280,140.840,397.599,169.226,43.530,158.189
C08822=1032.273,140.555,397.623,169.222,43.532,158.189
C08823=1032.267,140.270,397.648,169.219,43.533,158.189
C08824=1032.259,139.985,397.672,169.217,43.535,158.189
C08825=1032.254,139.736,397.694,169.214,43.536,158.189
C08826=1032.248,139.487,397.715,169.211,43.537,158.189
C08827=1032.242,139.237,397.736,169.209,43.539,158.190
C08828=1032.235,138.989,397.757,169.206,43.540,158.190
C08829=1032.229,138.740,397.779,169.203,43.541,158.190
C08830=1032.224,138.491,397.799,169.201,43.543,158.190
C08831=1032.218,138.242,397.821,169.198,43.544,158.190
C08832=1032.211,137.993,397.842,169.196,43.546,158.190
C08833=1032.205,137.744,397.863,169.193,43.547,158.190
C08834=1032.200,137.494,397.884,169.190,43.549,158.190
C08835=1032.193,137.245,397.905,169.188,43.550,158.190
C08836=1032.187,136.997,397.926,169.185,43.551,158.190
C08837=1032.181,136.747,397.947,169.182,43.553,158.190
C08838=1032.175,136.499,397.968,169.180,43.554,158.190
C08839=1032.169,136.250,397.990,169.178,43.556,158.191
C08840=1032.163,136.000,398.010,169.175,43.557,158.191
C08841=1032.157,135.752,398.031,169.172,43.559,158.191
C08842=1032.151,135.502,398.052,169.169,43.560,158.191
C08843=1032.145,135.253,398.073,169.167,43.562,158.191
C08844=1032.138,135.004,398.094,169.164,43.563,158.191
C08845=1032.132,134.755,398.115,169.162,43.564,158.191
C08846=1032.126,134.506,398.136,169.160,43.566,158.191
C08847=1032.120,134.257,398.157,169.157,43.568,158.191
C08848=1032.115,134.008,398.178,169.154,43.569,158.191
C08849=1032.108,133.759,398.199,169.151,43.571,158.191
C08850=1032.103,133.510,398.220,169.149,43.572,158.191
C08851=1032.096,133.261,398.241,169.147,43.573,158.191
C08852=1032.090,133.011,398.262,169.144,43.575,158.192
C08853=1032.084,132.763,398.283,169.141,43.576,158.192
C08854=1032.078,132.513,398.303,169.139,43.578,158.192
C08855=1032.072,132.265,398.325,169.136,43.580,158.192
C08856=1032.066,132.015,398.345,169.133,43.581,158.192
C08857=1032.060,131.767,398.366,169.132,43.582,158.192
C08858=1032.054,131.517,398.387,169.129,43.584,158.192
C08859=1032.048,131.269,398.408,169.126,43.585,158.192
C08860=1032.042,131.019,398.429,169.123,43.587,158.192
C08861=1032.036,130.771,398.449,169.120,43.588,158.192
C08862=1032.030,130.521,398.470,169.118,43.590,158.192
C08863=1032.024,130.272,398.490,169.116,43.591,158.192
C08864=1032.017,130.023,398.511,169.113,43.593,158.192
C08865=1032.012,129.774,398.532,169.111,43.594,158.193
C08866=1032.005,129.525,398.552,169.108,43.596,158.193
C08867=1031.998,129.276,398.573,169.105,43.598,158.193
C08868=1031.992,129.027,398.593,169.103,43.599,158.193
C08869=1031.986,128.777,398.614,169.100,43.601,158.193
C08870=1031.980,128.529,398.635,169.098,43.602,158.193
C08871=1031.973,128.279,398.655,169.096,43.603,158.193
C08872=1031.968,128.030,398.676,169.093,43.605,158.193
C08873=1031.962,127.781,398.696,169.090,43.607,158.193
C08874=1031.955,127.533,398.717,169.087,43.608,158.193
C08875=1031.949,127.283,398.737,169.085,43.610,158.193
C08876=1031.943,127.034,398.758,169.082,43.611,158.193
C08877=1031.937,126.784,398.778,169.080,43.613,158.194
C08878=1031.931,126.536,398.799,169.078,43.615,158.194
C08879=1031.924,126.287,398.819,169.075,43.616,158.194
C08880=1031.919,126.038,398.839,169.072,43.618,158.194
C08881=1031.912,125.788,398.860,169.070,43.619,158.194
C08882=1031.906,125.540,398.880,169.067,43.621,158.194
C08883=1031.900,125.291,398.900,169.065,43.622,158.194
C08884=1031.894,125.041,398.921,169.063,43.624,158.194
C08885=1031.886,124.756,398.944,169.060,43.626,158.194
C08886=1031.880,124.471,398.968,169.056,43.628,158.195
C08887=1031.873,124.186,398.991,169.053,43.629,158.195
C08888=1031.866,123.901,399.015,169.051,43.631,158.195
C08889=1031.860,123.652,399.035,169.048,43.633,158.195
C08890=1031.853,123.402,399.055,169.045,43.634,158.195
C08891=1031.847,123.154,399.075,169.043,43.636,158.195
C08892=1031.841,122.904,399.096,169.041,43.638,158.195
C08893=1031.835,122.655,399.116,169.038,43.639,158.195
C08894=1031.829,122.406,399.136,169.036,43.641,158.195
C08895=1031.822,122.157,399.157,169.033,43.642,158.195
C08896=1031.817,121.908,399.178,169.030,43.644,158.196
C08897=1031.811,121.659,399.198,169.029,43.645,158.196
C08898=1031.805,121.410,399.218,169.026,43.647,158.196
C08899=1031.799,121.161,399.238,169.023,43.648,158.196
C08900=1031.793,120.911,399.259,169.020,43.650,158.196
C08901=1031.787,120.662,399.279,169.019,43.651,158.196
C08902=1031.781,120.414,399.299,169.016,43.653,158.196
C08903=1031.774,120.164,399.319,169.013,43.654,158.196
C08904=1031.769,119.915,399.340,169.011,43.656,158.196
C08905=1031.763,119.666,399.360,169.008,43.658,158.196
C08906=1031.756,119.417,399.380,169.006,43.659,158.196
C08907=1031.750,119.168,399.400,169.004,43.660,158.197
C08908=1031.744,118.919,399.420,169.001,43.662,158.197
C08909=1031.738,118.669,399.441,168.998,43.663,158.197
C08910=1031.732,118.420,399.461,168.996,43.665,158.197
C08911=1031.726,118.171,399.481,168.994,43.666,158.197
C08912=1031.720,117.922,399.501,168.991,43.668,158.197
C08913=1031.715,117.673,399.521,168.988,43.669,158.197
C08914=1031.709,117.424,399.541,168.987,43.671,158.197
C08915=1031.702,117.174,399.562,168.984,43.672,158.197
C08916=1031.696,116.926,399.582,168.981,43.674,158.197
C08917=1031.690,116.677,399.602,168.978,43.675,158.197
C08918=1031.685,116.428,399.622,168.977,43.677,158.198
C08919=1031.678,116.178,399.643,168.974,43.678,158.198
C08920=1031.672,115.929,399.663,168.971,43.680,158.198
C08921=1031.666,115.681,399.682,168.969,43.681,158.198
C08922=1031.661,115.431,399.703,168.967,43.683,158.198
C08923=1031.654,115.182,399.723,168.964,43.684,158.198
C08924=1031.649,114.933,399.743,168.962,43.686,158.198
C08925=1031.643,114.684,399.763,168.960,43.687,158.198
C08926=1031.637,114.435,399.783,168.957,43.689,158.198
C08927=1031.631,114.185,399.803,168.954,43.690,158.198
C08928=1031.625,113.936,399.823,168.952,43.692,158.198
C08929=1031.619,113.687,399.843,168.950,43.693,158.198
C08930=1031.613,113.439,399.863,168.947,43.695,158.199
C08931=1031.607,113.189,399.883,168.944,43.696,158.199
C08932=1031.601,112.940,399.903,168.942,43.698,158.199
C08933=1031.595,112.691,399.923,168.940,43.699,158.199
C08934=1031.588,112.441,399.943,168.937,43.701,158.199
C08935=1031.582,112.192,399.962,168.935,43.703,158.199
C08936=1031.576,111.943,399.982,168.932,43.704,158.199
C08937=1031.570,111.694,400.002,168.930,43.706,158.199
C08938=1031.564,111.446,400.022,168.928,43.708,158.199
C08939=1031.558,111.195,400.042,168.925,43.709,158.199
C08940=1031.552,110.947,400.062,168.922,43.711,158.200
C08941=1031.546,110.698,400.082,168.921,43.712,158.200
C08942=1031.540,110.448,400.101,168.918,43.714,158.200
C08943=1031.534,110.199,400.121,168.915,43.715,158.200
C08944=1031.528,109.950,400.141,168.913,43.717,158.200
C08945=1031.521,109.701,400.160,168.911,43.718,158.200
C08946=1031.515,109.452,400.180,168.908,43.720,158.200
C08947=1031.509,109.202,400.200,168.906,43.722,158.200
C08948=1031.503,108.953,400.220,168.903,43.723,158.200
C08949=1031.496,108.668,400.242,168.900,43.725,158.200
C08950=1031.489,108.382,400.264,168.898,43.727,158.201
C08951=1031.481,108.097,400.287,168.895,43.729,158.201
C08952=1031.474,107.812,400.309,168.892,43.731,158.201
C08953=1031.468,107.563,400.328,168.890,43.733,158.201
C08954=1031.462,107.314,400.348,168.887,43.735,158.201
C08955=1031.456,107.064,400.368,168.884,43.736,158.201
C08956=1031.450,106.815,400.388,168.883,43.737,158.201
C08957=1031.444,106.566,400.406,168.880,43.739,158.202
C08958=1031.438,106.317,400.426,168.877,43.741,158.202
C08959=1031.432,106.068,400.446,168.875,43.742,158.202
C08960=1031.426,105.819,400.465,168.873,43.744,158.202
C08961=1031.419,105.569,400.484,168.870,43.745,158.202
C08962=1031.413,105.320,400.504,168.868,43.747,158.202
C08963=1031.407,105.071,400.524,168.865,43.749,158.202
C08964=1031.401,104.822,400.544,168.863,43.750,158.202
C08965=1031.395,104.573,400.562,168.861,43.752,158.202
C08966=1031.389,104.324,400.582,168.858,43.754,158.202
C08967=1031.383,104.074,400.602,168.855,43.756,158.203
C08968=1031.377,103.825,400.622,168.854,43.757,158.203
C08969=1031.370,103.576,400.640,168.851,43.759,158.203
C08970=1031.364,103.327,400.660,168.848,43.761,158.203
C08971=1031.359,103.078,400.680,168.847,43.762,158.203
C08972=1031.352,102.829,400.698,168.844,43.763,158.203
C08973=1031.346,102.580,400.718,168.841,43.765,158.203
C08974=1031.340,102.330,400.738,168.839,43.767,158.203
C08975=1031.334,102.082,400.757,168.837,43.768,158.203
C08976=1031.328,101.833,400.776,168.834,43.769,158.203
C08977=1031.322,101.582,400.796,168.831,43.771,158.204
C08978=1031.316,101.334,400.816,168.830,43.773,158.204
C08979=1031.310,101.084,400.835,168.827,43.774,158.204
C08980=1031.304,100.835,400.854,168.824,43.776,158.204
C08981=1031.298,100.586,400.874,168.822,43.778,158.204
C08982=1031.292,100.337,400.893,168.820,43.779,158.204
C08983=1031.286,100.087,400.912,168.817,43.781,158.204
C08984=1031.280,99.839,400.931,168.815,43.783,158.204
C08985=1031.274,99.589,400.951,168.813,43.784,158.204
C08986=1031.267,99.340,400.969,168.810,43.786,158.205
C08987=1031.262,99.091,400.989,168.808,43.788,158.205
C08988=1031.254,98.842,401.008,168.805,43.789,158.205
C08989=1031.248,98.593,401.027,168.803,43.790,158.205
C08990=1031.242,98.343,401.046,168.801,43.792,158.205
C08991=1031.236,98.094,401.065,168.798,43.794,158.205
C08992=1031.230,97.845,401.084,168.796,43.796,158.205
C08993=1031.223,97.596,401.103,168.794,43.798,158.206
C08994=1031.218,97.347,401.123,168.791,43.799,158.206
C08995=1031.211,97.097,401.141,168.789,43.801,158.206
C08996=1031.206,96.848,401.161,168.786,43.803,158.206
C08997=1031.199,96.599,401.179,168.784,43.804,158.206
C08998=1031.194,96.349,401.198,168.781,43.806,158.206
C08999=1031.187,96.101,401.218,168.779,43.808,158.206
C09000=1031.180,95.852,401.236,168.776,43.809,158.206
C09001=1031.175,95.602,401.256,168.775,43.811,158.206
C09002=1031.168,95.353,401.274,168.772,43.812,158.206
C09003=1031.163,95.104,401.294,168.769,43.814,158.207
C09004=1031.156,94.855,401.312,168.768,43.816,158.207
C09005=1031.150,94.605,401.331,168.765,43.818,158.207
C09006=1031.144,94.356,401.350,168.762,43.819,158.207
C09007=1031.138,94.107,401.369,168.760,43.821,158.207
C09008=1031.132,93.858,401.388,168.758,43.823,158.207
C09009=1031.125,93.609,401.407,168.755,43.824,158.207
C09010=1031.120,93.360,401.427,168.753,43.826,158.207
C09011=1031.113,93.111,401.445,168.751,43.827,158.208
C09012=1031.107,92.861,401.465,168.748,43.829,158.208
C09013=1031.101,92.576,401.486,168.746,43.831,158.208
C09014=1031.093,92.290,401.508,168.743,43.833,158.208
C09015=1031.086,92.005,401.530,168.741,43.835,158.208
C09016=1031.079,91.720,401.551,168.737,43.836,158.208
C09017=1031.073,91.470,401.569,168.735,43.838,158.208
C09018=1031.067,91.221,401.589,168.733,43.840,158.208
C09019=1031.061,90.972,401.607,168.730,43.842,158.209
C09020=1031.055,90.722,401.627,168.728,43.843,158.209
C09021=1031.049,90.473,401.645,168.726,43.845,158.209
C09022=1031.043,90.224,401.664,168.723,43.847,158.209
C09023=1031.037,89.975,401.683,168.721,43.848,158.209
C09024=1031.031,89.725,401.702,168.718,43.850,158.209
C09025=1031.024,89.476,401.721,168.716,43.851,158.209
C09026=1031.018,89.227,401.740,168.713,43.853,158.209
C09027=1031.012,88.978,401.758,168.712,43.855,158.210
C09028=1031.005,88.728,401.776,168.709,43.856,158.210
C09029=1031.000,88.480,401.794,168.706,43.858,158.210
C09030=1030.993,88.231,401.813,168.704,43.860,158.210
C09031=1030.988,87.981,401.832,168.702,43.862,158.210
C09032=1030.981,87.732,401.851,168.699,43.864,158.210
C09033=1030.975,87.483,401.870,168.697,43.865,158.210
C09034=1030.969,87.233,401.888,168.695,43.866,158.210
C09035=1030.962,86.984,401.906,168.692,43.868,158.210
C09036=1030.956,86.735,401.925,168.690,43.870,158.211
C09037=1030.949,86.486,401.944,168.687,43.872,158.211
C09038=1030.943,86.236,401.962,168.686,43.874,158.211
C09039=1030.937,85.987,401.981,168.683,43.876,158.211
C09040=1030.931,85.738,401.999,168.680,43.877,158.211
C09041=1030.925,85.489,402.018,168.678,43.879,158.211
C09042=1030.919,85.240,402.036,168.676,43.881,158.211
C09043=1030.913,84.990,402.054,168.673,43.882,158.211
C09044=1030.906,84.741,402.073,168.671,43.884,158.212
C09045=1030.900,84.492,402.092,168.669,43.885,158.212
C09046=1030.894,84.242,402.110,168.666,43.887,158.212
C09047=1030.888,83.993,402.129,168.664,43.889,158.212
C09048=1030.882,83.744,402.147,168.661,43.891,158.212
C09049=1030.876,83.495,402.166,168.659,43.892,158.212
C09050=1030.870,83.246,402.184,168.657,43.894,158.212
C09051=1030.863,82.997,402.202,168.654,43.896,158.212
C09052=1030.857,82.747,402.221,168.653,43.898,158.213
C09053=1030.851,82.498,402.239,168.650,43.899,158.213
C09054=1030.844,82.249,402.257,168.647,43.901,158.213
C09055=1030.839,81.999,402.277,168.646,43.902,158.213
C09056=1030.833,81.750,402.294,168.643,43.904,158.213
C09057=1030.827,81.501,402.313,168.640,43.906,158.213
C09058=1030.820,81.252,402.332,168.637,43.907,158.213
C09059=1030.814,81.002,402.350,168.636,43.909,158.213
C09060=1030.808,80.753,402.368,168.633,43.911,158.213
C09061=1030.802,80.505,402.386,168.631,43.913,158.214
C09062=1030.796,80.255,402.404,168.629,43.914,158.214
C09063=1030.789,80.006,402.423,168.626,43.916,158.214
C09064=1030.784,79.756,402.442,168.624,43.918,158.214
C09065=1030.777,79.506,402.460,168.622,43.919,158.214
C09066=1030.772,79.258,402.478,168.619,43.921,158.214
C09067=1030.766,79.008,402.496,168.617,43.923,158.214
C09068=1030.759,78.759,402.515,168.615,43.924,158.214
C09069=1030.753,78.509,402.533,168.612,43.926,158.215
C09070=1030.747,78.261,402.551,168.610,43.927,158.215
C09071=1030.741,78.011,402.569,168.608,43.929,158.215
C09072=1030.735,77.762,402.588,168.605,43.931,158.215
C09073=1030.728,77.512,402.606,168.603,43.933,158.215
C09074=1030.722,77.263,402.624,168.600,43.934,158.215
C09075=1030.717,77.014,402.642,168.598,43.936,158.215
C09076=1030.710,76.765,402.661,168.596,43.938,158.215
C09077=1030.703,76.480,402.681,168.593,43.940,158.215
C09078=1030.696,76.195,402.702,168.591,43.941,158.216
C09079=1030.689,75.908,402.723,168.588,43.943,158.216
C09080=1030.682,75.623,402.743,168.585,43.946,158.216
C09081=1030.676,75.374,402.762,168.583,43.947,158.216
C09082=1030.669,75.124,402.779,168.580,43.949,158.216
C09083=1030.663,74.876,402.797,168.578,43.951,158.216
C09084=1030.657,74.626,402.815,168.576,43.953,158.216
C09085=1030.651,74.377,402.833,168.573,43.955,158.217
C09086=1030.644,74.127,402.852,168.571,43.956,158.217
C09087=1030.639,73.878,402.870,168.568,43.958,158.217
C09088=1030.632,73.629,402.887,168.566,43.959,158.217
C09089=1030.625,73.380,402.906,168.564,43.961,158.217
C09090=1030.620,73.131,402.923,168.561,43.963,158.217
C09091=1030.614,72.881,402.941,168.560,43.965,158.217
C09092=1030.607,72.632,402.960,168.557,43.967,158.218
C09093=1030.601,72.382,402.978,168.554,43.968,158.218
C09094=1030.595,72.133,402.995,168.552,43.970,158.218
C09095=1030.589,71.884,403.013,168.550,43.972,158.218
C09096=1030.582,71.635,403.031,168.547,43.973,158.218
C09097=1030.577,71.386,403.049,168.545,43.975,158.218
C09098=1030.571,71.136,403.067,168.543,43.976,158.218
C09099=1030.564,70.887,403.085,168.540,43.978,158.218
C09100=1030.558,70.638,403.102,168.538,43.980,158.218
C09101=1030.552,70.388,403.120,168.536,43.982,158.219
C09102=1030.546,70.139,403.139,168.534,43.984,158.219
C09103=1030.539,69.890,403.156,168.531,43.985,158.219
